C09107=1059.255,344.994,392.279,173.812,36.431,156.854
C09108=1059.262,345.241,392.243,173.816,36.436,156.855
C09109=1059.268,345.487,392.207,173.819,36.441,156.856
C09110=1059.276,345.733,392.171,173.824,36.446,156.857
C09111=1059.282,345.979,392.135,173.828,36.451,156.859
C09112=1059.289,346.224,392.098,173.832,36.455,156.860
C09113=1059.296,346.470,392.063,173.836,36.460,156.861
C09114=1059.302,346.716,392.026,173.841,36.466,156.862
C09115=1059.308,346.961,391.990,173.844,36.471,156.863
C09116=1059.315,347.208,391.954,173.848,36.476,156.864
C09117=1059.323,347.455,391.918,173.853,36.480,156.865
C09118=1059.329,347.702,391.882,173.856,36.485,156.866
C09119=1059.336,347.950,391.845,173.861,36.490,156.868
C09120=1059.343,348.196,391.809,173.865,36.495,156.869
C09121=1059.350,348.444,391.772,173.869,36.500,156.870
C09122=1059.356,348.690,391.735,173.873,36.506,156.871
C09123=1059.363,348.938,391.698,173.878,36.511,156.872
C09124=1059.371,349.185,391.662,173.881,36.516,156.873
C09125=1059.377,349.433,391.626,173.886,36.521,156.875
C09126=1059.384,349.680,391.589,173.890,36.526,156.876
C09127=1059.391,349.928,391.552,173.895,36.531,156.877
C09128=1059.398,350.174,391.517,173.898,36.536,156.878
C09129=1059.405,350.421,391.479,173.903,36.541,156.879
C09130=1059.411,350.668,391.443,173.907,36.547,156.881
C09131=1059.418,350.916,391.406,173.911,36.552,156.882
C09132=1059.425,351.163,391.370,173.916,36.557,156.883
C09133=1059.433,351.410,391.332,173.920,36.562,156.884
C09134=1059.439,351.657,391.296,173.925,36.567,156.885
C09135=1059.446,351.905,391.259,173.928,36.572,156.886
C09136=1059.453,352.151,391.222,173.933,36.578,156.888
C09137=1059.459,352.399,391.185,173.937,36.583,156.889
C09138=1059.466,352.647,391.148,173.941,36.588,156.890
C09139=1059.473,352.893,391.111,173.945,36.593,156.891
C09140=1059.480,353.141,391.074,173.950,36.598,156.893
C09141=1059.487,353.387,391.037,173.955,36.603,156.894
C09142=1059.494,353.635,391.000,173.959,36.609,156.895
C09143=1059.500,353.882,390.963,173.963,36.614,156.896
C09144=1059.507,354.129,390.926,173.967,36.619,156.897
C09145=1059.514,354.377,390.889,173.972,36.625,156.899
C09146=1059.521,354.623,390.852,173.976,36.630,156.900
C09147=1059.528,354.871,390.815,173.980,36.635,156.901
C09148=1059.535,355.118,390.777,173.985,36.640,156.902
C09149=1059.542,355.364,390.740,173.989,36.646,156.904
C09150=1059.549,355.612,390.703,173.994,36.651,156.905
C09151=1059.556,355.859,390.666,173.998,36.656,156.906
C09152=1059.563,356.106,390.629,174.002,36.662,156.907
C09153=1059.570,356.353,390.592,174.007,36.667,156.909
C09154=1059.577,356.601,390.554,174.012,36.672,156.910
C09155=1059.584,356.848,390.517,174.015,36.678,156.911
C09156=1059.591,357.094,390.480,174.020,36.683,156.912
C09157=1059.598,357.342,390.443,174.025,36.688,156.914
C09158=1059.605,357.589,390.405,174.029,36.694,156.915
C09159=1059.612,357.836,390.368,174.033,36.699,156.916
C09160=1059.619,358.083,390.330,174.038,36.705,156.917
C09161=1059.626,358.330,390.293,174.042,36.710,156.919
C09162=1059.633,358.577,390.256,174.047,36.715,156.920
C09163=1059.640,358.824,390.217,174.052,36.721,156.921
C09164=1059.647,359.071,390.180,174.056,36.726,156.923
C09165=1059.654,359.320,390.142,174.060,36.732,156.924
C09166=1059.661,359.569,390.104,174.065,36.737,156.925
C09167=1059.667,359.818,390.067,174.070,36.743,156.927
C09168=1059.675,360.067,390.028,174.074,36.749,156.928
C09169=1059.682,360.313,389.991,174.079,36.754,156.929
C09170=1059.689,360.560,389.953,174.083,36.760,156.930
C09171=1059.696,360.807,389.916,174.087,36.765,156.932
C09172=1059.703,361.055,389.877,174.092,36.770,156.933
C09173=1059.710,361.302,389.840,174.097,36.776,156.934
C09174=1059.717,361.549,389.802,174.102,36.781,156.936
C09175=1059.725,361.796,389.764,174.106,36.787,156.937
C09176=1059.731,362.043,389.726,174.110,36.793,156.938
C09177=1059.739,362.290,389.689,174.115,36.799,156.940
C09178=1059.746,362.536,389.651,174.120,36.804,156.941
C09179=1059.752,362.783,389.613,174.124,36.810,156.942
C09180=1059.759,363.031,389.575,174.129,36.815,156.944
C09181=1059.767,363.277,389.537,174.134,36.821,156.945
C09182=1059.773,363.525,389.499,174.139,36.826,156.946
C09183=1059.781,363.772,389.461,174.143,36.832,156.948
C09184=1059.788,364.018,389.423,174.147,36.838,156.949
C09185=1059.795,364.266,389.385,174.152,36.844,156.950
C09186=1059.802,364.512,389.346,174.157,36.849,156.952
C09187=1059.809,364.760,389.308,174.162,36.855,156.953
C09188=1059.815,365.006,389.270,174.166,36.861,156.954
C09189=1059.823,365.253,389.231,174.171,36.866,156.956
C09190=1059.830,365.500,389.193,174.176,36.873,156.957
C09191=1059.837,365.747,389.155,174.180,36.878,156.959
C09192=1059.844,365.994,389.116,174.185,36.884,156.960
C09193=1059.851,366.241,389.079,174.190,36.890,156.961
C09194=1059.858,366.488,389.040,174.194,36.896,156.963
C09195=1059.866,366.734,389.001,174.199,36.901,156.964
C09196=1059.873,366.982,388.963,174.204,36.907,156.966
C09197=1059.879,367.229,388.924,174.209,36.913,156.967
C09198=1059.887,367.476,388.886,174.214,36.919,156.968
C09199=1059.894,367.722,388.847,174.219,36.925,156.970
C09200=1059.901,367.969,388.809,174.223,36.931,156.971
C09201=1059.908,368.216,388.770,174.228,36.937,156.973
C09202=1059.915,368.463,388.732,174.232,36.942,156.974
C09203=1059.922,368.710,388.694,174.237,36.948,156.975
C09204=1059.930,368.957,388.654,174.242,36.954,156.977
C09205=1059.936,369.204,388.616,174.247,36.960,156.978
C09206=1059.944,369.451,388.577,174.252,36.966,156.980
C09207=1059.951,369.697,388.539,174.257,36.972,156.981
C09208=1059.958,369.944,388.500,174.262,36.978,156.983
C09209=1059.966,370.192,388.461,174.267,36.984,156.984
C09210=1059.973,370.438,388.422,174.271,36.990,156.985
C09211=1059.980,370.684,388.383,174.276,36.996,156.987
C09212=1059.987,370.931,388.344,174.281,37.002,156.988
C09213=1059.995,371.179,388.305,174.286,37.008,156.990
C09214=1060.002,371.425,388.267,174.291,37.014,156.991
C09215=1060.009,371.672,388.228,174.296,37.020,156.993
C09216=1060.016,371.919,388.189,174.301,37.026,156.994
C09217=1060.024,372.165,388.150,174.306,37.032,156.996
C09218=1060.031,372.412,388.111,174.311,37.038,156.997
C09219=1060.039,372.660,388.072,174.316,37.044,156.999
C09220=1060.046,372.906,388.032,174.321,37.050,157.000
C09221=1060.053,373.173,387.990,174.326,37.057,157.002
C09222=1060.060,373.440,387.948,174.332,37.064,157.003
C09223=1060.069,373.707,387.906,174.337,37.071,157.005
C09224=1060.077,373.974,387.863,174.342,37.077,157.007
C09225=1060.084,374.221,387.824,174.347,37.083,157.008
C09226=1060.091,374.468,387.785,174.352,37.090,157.010
C09227=1060.098,374.714,387.745,174.357,37.096,157.011
C09228=1060.106,374.962,387.706,174.362,37.102,157.013
C09229=1060.113,375.208,387.666,174.367,37.109,157.014
C09230=1060.120,375.454,387.627,174.372,37.115,157.016
C09231=1060.127,375.702,387.588,174.377,37.121,157.017
C09232=1060.134,375.948,387.548,174.382,37.127,157.019
C09233=1060.142,376.195,387.509,174.388,37.134,157.020
C09234=1060.149,376.442,387.469,174.394,37.140,157.022
C09235=1060.157,376.689,387.429,174.399,37.146,157.023
C09236=1060.164,376.935,387.390,174.404,37.152,157.025
C09237=1060.171,377.182,387.351,174.409,37.159,157.027
C09238=1060.178,377.429,387.311,174.414,37.166,157.028
C09239=1060.186,377.675,387.271,174.419,37.172,157.030
C09240=1060.193,377.922,387.232,174.424,37.178,157.031
C09241=1060.201,378.169,387.192,174.429,37.185,157.033
C09242=1060.208,378.415,387.152,174.434,37.191,157.034
C09243=1060.216,378.662,387.112,174.439,37.197,157.036
C09244=1060.223,378.908,387.073,174.444,37.204,157.038
C09245=1060.231,379.155,387.033,174.451,37.211,157.039
C09246=1060.238,379.402,386.993,174.456,37.217,157.041
C09247=1060.245,379.648,386.953,174.461,37.223,157.042
C09248=1060.253,379.895,386.913,174.466,37.230,157.044
C09249=1060.261,380.142,386.873,174.471,37.236,157.045
C09250=1060.267,380.388,386.833,174.476,37.243,157.047
C09251=1060.275,380.635,386.793,174.482,37.249,157.049
C09252=1060.283,380.882,386.753,174.487,37.256,157.050
C09253=1060.290,381.128,386.714,174.492,37.262,157.052
C09254=1060.297,381.375,386.673,174.498,37.270,157.054
C09255=1060.304,381.621,386.633,174.503,37.276,157.055
C09256=1060.312,381.868,386.593,174.508,37.283,157.057
C09257=1060.319,382.114,386.552,174.514,37.289,157.059
C09258=1060.326,382.361,386.512,174.519,37.296,157.060
C09259=1060.334,382.608,386.472,174.524,37.303,157.062
C09260=1060.341,382.854,386.431,174.530,37.309,157.064
C09261=1060.349,383.101,386.391,174.535,37.316,157.065
C09262=1060.356,383.347,386.351,174.541,37.323,157.067
C09263=1060.363,383.594,386.311,174.546,37.330,157.069
C09264=1060.371,383.840,386.270,174.551,37.337,157.070
C09265=1060.378,384.087,386.229,174.557,37.344,157.072
C09266=1060.386,384.333,386.189,174.562,37.350,157.074
C09267=1060.394,384.580,386.149,174.568,37.357,157.075
C09268=1060.401,384.826,386.108,174.573,37.364,157.077
C09269=1060.409,385.073,386.067,174.578,37.371,157.079
C09270=1060.417,385.320,386.027,174.585,37.378,157.081
C09271=1060.424,385.566,385.986,174.590,37.384,157.082
C09272=1060.431,385.812,385.946,174.595,37.391,157.084
C09273=1060.438,386.059,385.905,174.600,37.398,157.086
C09274=1060.446,386.305,385.865,174.607,37.405,157.087
C09275=1060.454,386.552,385.824,174.612,37.412,157.089
C09276=1060.462,386.798,385.783,174.617,37.419,157.091
C09277=1060.471,387.097,385.733,174.625,37.428,157.093
C09278=1060.481,387.395,385.684,174.631,37.436,157.095
C09279=1060.490,387.693,385.635,174.638,37.445,157.097
C09280=1060.499,387.992,385.585,174.644,37.453,157.099
C09281=1060.507,388.238,385.545,174.650,37.460,157.101
C09282=1060.514,388.484,385.503,174.656,37.467,157.103
C09283=1060.522,388.731,385.463,174.661,37.474,157.105
C09284=1060.529,388.977,385.421,174.667,37.481,157.107
C09285=1060.537,389.224,385.381,174.673,37.488,157.108
C09286=1060.545,389.470,385.340,174.679,37.495,157.110
C09287=1060.553,389.716,385.299,174.684,37.502,157.112
C09288=1060.560,389.962,385.257,174.691,37.509,157.114
C09289=1060.568,390.209,385.216,174.696,37.517,157.116
C09290=1060.576,390.455,385.175,174.701,37.524,157.117
C09291=1060.583,390.702,385.134,174.708,37.531,157.119
C09292=1060.592,390.948,385.092,174.713,37.539,157.121
C09293=1060.599,391.195,385.051,174.719,37.546,157.123
C09294=1060.606,391.441,385.010,174.725,37.553,157.125
C09295=1060.615,391.687,384.968,174.731,37.560,157.126
C09296=1060.622,391.934,384.927,174.737,37.568,157.128
C09297=1060.630,392.180,384.885,174.742,37.575,157.130
C09298=1060.637,392.426,384.844,174.748,37.582,157.132
C09299=1060.646,392.673,384.802,174.754,37.590,157.134
C09300=1060.653,392.919,384.761,174.760,37.597,157.136
C09301=1060.661,393.165,384.719,174.765,37.604,157.138
C09302=1060.668,393.412,384.678,174.772,37.612,157.140
C09303=1060.676,393.658,384.636,174.777,37.620,157.141
C09304=1060.684,393.904,384.594,174.784,37.627,157.143
C09305=1060.692,394.150,384.552,174.790,37.635,157.145
C09306=1060.699,394.397,384.511,174.796,37.642,157.147
C09307=1060.707,394.643,384.469,174.802,37.650,157.149
C09308=1060.715,394.889,384.427,174.807,37.657,157.151
C09309=1060.723,395.135,384.385,174.814,37.665,157.153
C09310=1060.730,395.382,384.344,174.819,37.672,157.155
C09311=1060.738,395.629,384.301,174.826,37.680,157.157
C09312=1060.746,395.875,384.259,174.831,37.688,157.159
C09313=1060.753,396.121,384.217,174.838,37.695,157.161
C09314=1060.762,396.367,384.175,174.844,37.703,157.163
C09315=1060.769,396.613,384.133,174.850,37.711,157.165
C09316=1060.777,396.860,384.091,174.856,37.718,157.167
C09317=1060.786,397.106,384.050,174.862,37.726,157.169
C09318=1060.794,397.352,384.007,174.868,37.734,157.171
C09319=1060.801,397.598,383.965,174.875,37.741,157.173
C09320=1060.809,397.845,383.922,174.880,37.749,157.175
C09321=1060.817,398.091,383.880,174.887,37.758,157.177
C09322=1060.825,398.337,383.837,174.892,37.765,157.179
C09323=1060.833,398.583,383.795,174.899,37.773,157.181
C09324=1060.841,398.830,383.753,174.906,37.781,157.183
C09325=1060.849,399.075,383.710,174.911,37.789,157.185
C09326=1060.857,399.322,383.668,174.918,37.797,157.187
C09327=1060.864,399.568,383.626,174.924,37.805,157.189
C09328=1060.872,399.814,383.583,174.931,37.813,157.191
C09329=1060.880,400.060,383.541,174.937,37.821,157.193
C09330=1060.888,400.306,383.498,174.943,37.829,157.195
C09331=1060.897,400.553,383.455,174.950,37.837,157.197
C09332=1060.905,400.798,383.413,174.955,37.845,157.199
C09333=1060.915,401.114,383.358,174.963,37.855,157.202
C09334=1060.925,401.430,383.304,174.973,37.865,157.205
C09335=1060.935,401.745,383.248,174.981,37.876,157.207
C09336=1060.946,402.060,383.194,174.989,37.886,157.210
C09337=1060.953,402.307,383.151,174.995,37.894,157.212
C09338=1060.962,402.553,383.108,175.001,37.902,157.214
C09339=1060.970,402.798,383.065,175.008,37.911,157.216
C09340=1060.977,403.045,383.022,175.014,37.919,157.219
C09341=1060.986,403.291,382.979,175.021,37.927,157.221
C09342=1060.994,403.537,382.936,175.028,37.935,157.223
C09343=1061.002,403.784,382.892,175.034,37.944,157.225
C09344=1061.010,404.029,382.850,175.040,37.952,157.227
C09345=1061.018,404.275,382.806,175.047,37.960,157.229
C09346=1061.026,404.521,382.763,175.054,37.969,157.232
C09347=1061.035,404.767,382.720,175.061,37.977,157.234
C09348=1061.042,405.014,382.676,175.067,37.986,157.236
C09349=1061.051,405.260,382.633,175.074,37.994,157.238
C09350=1061.059,405.506,382.590,175.080,38.002,157.240
C09351=1061.067,405.752,382.547,175.086,38.011,157.243
C09352=1061.075,405.999,382.503,175.093,38.020,157.245
C09353=1061.083,406.244,382.459,175.100,38.028,157.247
C09354=1061.092,406.490,382.416,175.107,38.037,157.249
C09355=1061.099,406.737,382.372,175.114,38.045,157.252
C09356=1061.107,406.982,382.328,175.121,38.054,157.254
C09357=1061.116,407.229,382.285,175.127,38.063,157.256
C09358=1061.124,407.475,382.241,175.134,38.071,157.259
C09359=1061.132,407.720,382.197,175.141,38.080,157.261
C09360=1061.140,407.967,382.154,175.148,38.089,157.263
C09361=1061.148,408.212,382.109,175.155,38.097,157.265
C09362=1061.157,408.458,382.066,175.162,38.106,157.268
C09363=1061.165,408.704,382.022,175.169,38.115,157.270
C09364=1061.173,408.951,381.978,175.175,38.123,157.272
C09365=1061.181,409.196,381.935,175.182,38.132,157.275
C09366=1061.190,409.442,381.890,175.189,38.141,157.277
C09367=1061.198,409.689,381.846,175.196,38.150,157.280
C09368=1061.206,409.935,381.802,175.203,38.159,157.282
C09369=1061.215,410.180,381.758,175.210,38.168,157.284
C09370=1061.223,410.426,381.714,175.217,38.177,157.287
C09371=1061.231,410.672,381.670,175.225,38.186,157.289
C09372=1061.240,410.918,381.626,175.232,38.195,157.291
C09373=1061.248,411.164,381.582,175.239,38.204,157.294
C09374=1061.256,411.410,381.538,175.246,38.213,157.296
C09375=1061.265,411.656,381.493,175.253,38.222,157.299
C09376=1061.274,411.902,381.449,175.260,38.231,157.301
C09377=1061.282,412.147,381.405,175.268,38.240,157.303
C09378=1061.290,412.394,381.360,175.275,38.249,157.306
C09379=1061.298,412.640,381.316,175.282,38.258,157.308
C09380=1061.308,412.886,381.272,175.289,38.267,157.311
C09381=1061.316,413.131,381.227,175.296,38.277,157.313
C09382=1061.324,413.377,381.182,175.304,38.286,157.316
C09383=1061.333,413.623,381.138,175.311,38.295,157.318
C09384=1061.342,413.868,381.094,175.318,38.304,157.321
C09385=1061.350,414.115,381.049,175.326,38.314,157.323
C09386=1061.359,414.360,381.004,175.333,38.323,157.326
C09387=1061.368,414.606,380.959,175.341,38.332,157.328
C09388=1061.376,414.852,380.914,175.348,38.342,157.331
C09389=1061.389,415.252,380.841,175.360,38.357,157.335
C09390=1061.404,415.652,380.768,175.373,38.373,157.339
C09391=1061.417,416.053,380.695,175.385,38.388,157.343
C09392=1061.431,416.453,380.621,175.397,38.404,157.348
C09393=1061.439,416.698,380.576,175.405,38.413,157.350
C09394=1061.448,416.943,380.531,175.412,38.423,157.353
C09395=1061.457,417.189,380.486,175.420,38.432,157.355
C09396=1061.465,417.435,380.441,175.428,38.442,157.358
C09397=1061.474,417.681,380.396,175.435,38.452,157.361
C09398=1061.483,417.927,380.350,175.443,38.462,157.363
C09399=1061.492,418.172,380.305,175.450,38.472,157.366
C09400=1061.501,418.418,380.260,175.459,38.481,157.369
C09401=1061.509,418.664,380.214,175.466,38.491,157.371
C09402=1061.518,418.910,380.168,175.474,38.501,157.374
C09403=1061.526,419.155,380.123,175.482,38.511,157.377
C09404=1061.535,419.401,380.078,175.490,38.520,157.379
C09405=1061.544,419.646,380.032,175.498,38.530,157.382
C09406=1061.554,419.892,379.986,175.506,38.540,157.385
C09407=1061.562,420.138,379.940,175.514,38.551,157.388
C09408=1061.571,420.384,379.895,175.521,38.561,157.390
C09409=1061.585,420.795,379.818,175.535,38.577,157.395
C09410=1061.600,421.207,379.741,175.548,38.594,157.400
C09411=1061.615,421.618,379.664,175.563,38.611,157.404
C09412=1061.629,422.030,379.587,175.576,38.629,157.409
C09413=1061.639,422.275,379.541,175.584,38.639,157.412
C09414=1061.647,422.521,379.495,175.593,38.649,157.415
C09415=1061.656,422.767,379.449,175.600,38.660,157.418
C09416=1061.665,423.012,379.402,175.609,38.670,157.421
C09417=1061.674,423.258,379.356,175.617,38.680,157.424
C09418=1061.683,423.504,379.310,175.626,38.691,157.426
C09419=1061.692,423.750,379.263,175.633,38.701,157.429
C09420=1061.701,423.995,379.217,175.642,38.711,157.432
C09421=1061.710,424.240,379.170,175.651,38.722,157.435
C09422=1061.719,424.486,379.124,175.659,38.733,157.438
C09423=1061.728,424.731,379.077,175.668,38.743,157.441
C09424=1061.737,424.976,379.031,175.675,38.754,157.444
C09425=1061.747,425.222,378.985,175.684,38.765,157.447
C09426=1061.755,425.468,378.938,175.693,38.775,157.450
C09427=1061.765,425.713,378.892,175.701,38.786,157.453
C09428=1061.773,425.958,378.845,175.710,38.797,157.456
C09429=1061.783,426.204,378.798,175.719,38.807,157.459
C09430=1061.792,426.449,378.751,175.727,38.818,157.462
C09431=1061.801,426.695,378.704,175.736,38.828,157.465
C09432=1061.811,426.940,378.657,175.745,38.839,157.468
C09433=1061.819,427.185,378.611,175.754,38.851,157.471
C09434=1061.828,427.432,378.563,175.762,38.861,157.474
C09435=1061.838,427.676,378.517,175.771,38.872,157.477
C09436=1061.847,427.921,378.469,175.780,38.884,157.480
C09437=1061.856,428.167,378.422,175.789,38.894,157.483
C09438=1061.865,428.412,378.375,175.798,38.906,157.487
C09439=1061.875,428.658,378.327,175.806,38.916,157.490
C09440=1061.884,428.903,378.281,175.815,38.928,157.493
C09441=1061.897,429.244,378.215,175.828,38.943,157.497
C09442=1061.909,429.585,378.149,175.840,38.959,157.502
C09443=1061.923,429.926,378.083,175.853,38.974,157.506
C09444=1061.935,430.266,378.017,175.865,38.990,157.511
C09445=1061.945,430.512,377.969,175.875,39.001,157.514
C09446=1061.954,430.758,377.922,175.884,39.013,157.517
C09447=1061.963,431.002,377.874,175.893,39.024,157.520
C09448=1061.972,431.248,377.826,175.902,39.036,157.524
C09449=1061.982,431.494,377.778,175.911,39.047,157.527
C09450=1061.991,431.738,377.730,175.921,39.059,157.530
C09451=1062.001,431.984,377.682,175.931,39.070,157.534
C09452=1062.010,432.229,377.635,175.940,39.082,157.537
C09453=1062.019,432.473,377.587,175.950,39.093,157.540
C09454=1062.029,432.719,377.539,175.959,39.105,157.543
C09455=1062.038,432.964,377.490,175.968,39.117,157.547
C09456=1062.048,433.210,377.442,175.978,39.128,157.550
C09457=1062.058,433.455,377.394,175.987,39.141,157.554
C09458=1062.067,433.699,377.346,175.996,39.152,157.557
C09459=1062.076,433.944,377.298,176.007,39.164,157.560
C09460=1062.086,434.189,377.249,176.016,39.176,157.564
C09461=1062.096,434.434,377.201,176.026,39.188,157.567
C09462=1062.105,434.679,377.152,176.035,39.200,157.571
C09463=1062.115,434.925,377.104,176.046,39.212,157.574
C09464=1062.125,435.170,377.056,176.055,39.224,157.578
C09465=1062.134,435.415,377.007,176.065,39.236,157.581
C09466=1062.143,435.660,376.958,176.074,39.248,157.585
C09467=1062.153,435.905,376.910,176.085,39.260,157.588
C09468=1062.163,436.150,376.861,176.095,39.272,157.592
C09469=1062.173,436.395,376.813,176.105,39.285,157.595
C09470=1062.183,436.639,376.763,176.115,39.297,157.599
C09471=1062.193,436.884,376.715,176.125,39.309,157.603
C09472=1062.202,437.129,376.666,176.135,39.321,157.606
C09473=1062.213,437.375,376.618,176.145,39.334,157.610
C09474=1062.223,437.619,376.568,176.156,39.346,157.613
C09475=1062.232,437.865,376.519,176.165,39.359,157.617
C09476=1062.242,438.109,376.470,176.176,39.371,157.621
C09477=1062.252,438.355,376.421,176.186,39.384,157.624
C09478=1062.262,438.599,376.371,176.197,39.396,157.628
C09479=1062.271,438.844,376.323,176.206,39.409,157.632
C09480=1062.281,439.089,376.273,176.217,39.422,157.636
C09481=1062.291,439.334,376.223,176.227,39.434,157.639
C09482=1062.301,439.578,376.174,176.238,39.447,157.643
C09483=1062.311,439.823,376.125,176.249,39.460,157.647
C09484=1062.321,440.069,376.075,176.259,39.472,157.651
C09485=1062.331,440.313,376.026,176.270,39.485,157.654
C09486=1062.341,440.558,375.976,176.281,39.498,157.658
C09487=1062.351,440.803,375.927,176.291,39.511,157.662
C09488=1062.361,441.047,375.877,176.301,39.524,157.666
C09489=1062.371,441.292,375.826,176.312,39.537,157.670
C09490=1062.381,441.536,375.777,176.323,39.550,157.674
C09491=1062.391,441.782,375.727,176.335,39.564,157.678
C09492=1062.401,442.026,375.678,176.346,39.577,157.682
C09493=1062.412,442.271,375.627,176.356,39.590,157.686
C09494=1062.422,442.516,375.577,176.367,39.603,157.690
C09495=1062.432,442.760,375.527,176.378,39.616,157.693
C09496=1062.443,443.005,375.477,176.389,39.630,157.698
C09497=1062.453,443.260,375.424,176.400,39.644,157.702
C09498=1062.464,443.514,375.372,176.413,39.658,157.706
C09499=1062.474,443.769,375.319,176.424,39.672,157.710
C09500=1062.486,444.024,375.267,176.436,39.685,157.714
C09501=1062.495,444.268,375.217,176.447,39.699,157.718
C09502=1062.505,444.513,375.166,176.459,39.713,157.723
C09503=1062.516,444.758,375.116,176.470,39.726,157.727
C09504=1062.526,445.002,375.065,176.481,39.740,157.731
C09505=1062.537,445.247,375.014,176.493,39.754,157.735
C09506=1062.548,445.492,374.964,176.505,39.767,157.739
C09507=1062.557,445.736,374.913,176.516,39.781,157.743
C09508=1062.567,445.980,374.862,176.528,39.795,157.748
C09509=1062.579,446.224,374.811,176.539,39.809,157.752
C09510=1062.589,446.469,374.760,176.552,39.823,157.756
C09511=1062.599,446.714,374.709,176.563,39.837,157.760
C09512=1062.610,446.957,374.658,176.575,39.851,157.765
C09513=1062.621,447.202,374.607,176.587,39.865,157.769
C09514=1062.632,447.445,374.556,176.599,39.879,157.773
C09515=1062.643,447.689,374.506,176.610,39.893,157.777
C09516=1062.655,447.933,374.457,176.622,39.907,157.782
C09517=1062.668,448.177,374.406,176.635,39.920,157.786
C09518=1062.683,448.421,374.358,176.647,39.933,157.790
C09519=1062.697,448.665,374.311,176.659,39.946,157.794
C09520=1062.714,448.910,374.263,176.672,39.958,157.798
C09521=1062.730,449.155,374.217,176.684,39.971,157.802
C09522=1062.749,449.400,374.170,176.697,39.983,157.806
C09523=1062.767,449.646,374.125,176.710,39.994,157.809
C09524=1062.788,449.891,374.081,176.722,40.006,157.813
C09525=1062.452,449.899,373.808,176.715,40.125,157.846
C09526=1062.433,449.654,373.853,176.702,40.114,157.842
C09527=1062.414,449.409,373.898,176.689,40.102,157.838
C09528=1062.395,449.163,373.944,176.677,40.090,157.834
C09529=1062.379,448.919,373.990,176.664,40.078,157.830
C09530=1062.362,448.673,374.037,176.652,40.065,157.826
C09531=1062.347,448.429,374.086,176.639,40.052,157.822
C09532=1062.332,448.185,374.134,176.627,40.039,157.818
C09533=1062.319,447.941,374.183,176.615,40.026,157.814
C09534=1062.307,447.697,374.233,176.602,40.013,157.810
C09535=1062.295,447.453,374.283,176.591,39.999,157.806
C09536=1062.284,447.210,374.334,176.578,39.985,157.801
C09537=1062.274,446.967,374.385,176.567,39.971,157.797
C09538=1062.263,446.723,374.436,176.555,39.957,157.793
C09539=1062.252,446.478,374.487,176.542,39.943,157.789
C09540=1062.242,446.233,374.538,176.531,39.929,157.784
C09541=1062.231,445.989,374.589,176.519,39.916,157.780
C09542=1062.221,445.745,374.640,176.507,39.902,157.776
C09543=1062.210,445.500,374.691,176.496,39.888,157.772
C09544=1062.199,445.256,374.742,176.484,39.874,157.767
C09545=1062.189,445.011,374.792,176.473,39.860,157.763
C09546=1062.179,444.771,374.842,176.462,39.847,157.759
C09547=1062.169,444.530,374.892,176.449,39.834,157.755
C09548=1062.158,444.290,374.941,176.438,39.820,157.751
C09549=1062.148,444.050,374.991,176.427,39.807,157.747
C09550=1062.138,443.810,375.041,176.416,39.794,157.743
C09551=1062.128,443.570,375.090,176.405,39.780,157.739
C09552=1062.118,443.331,375.139,176.394,39.767,157.735
C09553=1062.108,443.091,375.189,176.383,39.754,157.731
C09554=1062.097,442.846,375.240,176.371,39.741,157.727
C09555=1062.087,442.602,375.289,176.360,39.728,157.723
C09556=1062.077,442.357,375.340,176.349,39.715,157.719
C09557=1062.067,442.112,375.389,176.339,39.702,157.715
C09558=1062.057,441.867,375.440,176.328,39.688,157.711
C09559=1062.046,441.623,375.490,176.317,39.675,157.707
C09560=1062.037,441.378,375.540,176.306,39.662,157.703
C09561=1062.026,441.133,375.589,176.295,39.649,157.699
C09562=1062.017,440.888,375.639,176.284,39.636,157.695
C09563=1062.006,440.643,375.689,176.273,39.624,157.692
C09564=1061.996,440.400,375.739,176.263,39.610,157.688
C09565=1061.986,440.154,375.789,176.252,39.597,157.684
C09566=1061.976,439.910,375.838,176.241,39.585,157.680
C09567=1061.966,439.664,375.888,176.230,39.572,157.676
C09568=1061.956,439.419,375.937,176.220,39.559,157.673
C09569=1061.946,439.175,375.986,176.209,39.547,157.669
C09570=1061.936,438.930,376.036,176.199,39.534,157.665
C09571=1061.926,438.685,376.086,176.189,39.522,157.661
C09572=1061.916,438.440,376.134,176.178,39.509,157.658
C09573=1061.906,438.195,376.184,176.167,39.496,157.654
C09574=1061.897,437.950,376.233,176.157,39.484,157.650
C09575=1061.887,437.706,376.282,176.147,39.471,157.646
C09576=1061.877,437.461,376.331,176.137,39.459,157.643
C09577=1061.867,437.215,376.381,176.126,39.447,157.639
C09578=1061.857,436.970,376.429,176.116,39.434,157.636
C09579=1061.847,436.725,376.478,176.106,39.422,157.632
C09580=1061.837,436.481,376.527,176.096,39.410,157.629
C09581=1061.828,436.236,376.576,176.085,39.398,157.625
C09582=1061.818,435.991,376.624,176.076,39.386,157.621
C09583=1061.808,435.746,376.673,176.066,39.374,157.618
C09584=1061.798,435.501,376.722,176.056,39.362,157.614
C09585=1061.788,435.256,376.770,176.046,39.350,157.611
C09586=1061.778,435.011,376.819,176.035,39.337,157.607
C09587=1061.768,434.766,376.867,176.026,39.326,157.604
C09588=1061.759,434.521,376.916,176.016,39.314,157.600
C09589=1061.749,434.276,376.964,176.007,39.302,157.597
C09590=1061.741,434.030,377.012,175.996,39.290,157.593
C09591=1061.731,433.786,377.061,175.987,39.278,157.590
C09592=1061.721,433.541,377.109,175.978,39.266,157.587
C09593=1061.711,433.296,377.158,175.968,39.255,157.583
C09594=1061.702,433.050,377.206,175.958,39.243,157.580
C09595=1061.692,432.805,377.254,175.948,39.231,157.576
C09596=1061.683,432.560,377.302,175.939,39.220,157.573
C09597=1061.674,432.315,377.350,175.930,39.208,157.570
C09598=1061.664,432.070,377.398,175.920,39.196,157.566
C09599=1061.654,431.825,377.447,175.911,39.185,157.563
C09600=1061.646,431.580,377.494,175.901,39.173,157.560
C09601=1061.636,431.334,377.542,175.892,39.161,157.556
C09602=1061.627,431.088,377.590,175.882,39.150,157.553
C09603=1061.618,430.844,377.638,175.873,39.139,157.550
C09604=1061.608,430.599,377.686,175.864,39.127,157.546
C09605=1061.598,430.353,377.733,175.855,39.116,157.543
C09606=1061.586,430.010,377.799,175.842,39.100,157.539
C09607=1061.573,429.668,377.866,175.829,39.085,157.534
C09608=1061.560,429.325,377.932,175.817,39.069,157.530
C09609=1061.547,428.982,377.998,175.804,39.054,157.525
C09610=1061.537,428.737,378.045,175.795,39.042,157.522
C09611=1061.528,428.492,378.093,175.786,39.031,157.519
C09612=1061.518,428.246,378.141,175.777,39.020,157.516
C09613=1061.510,428.001,378.187,175.768,39.010,157.513
C09614=1061.499,427.755,378.235,175.759,38.998,157.510
C09615=1061.491,427.510,378.281,175.750,38.987,157.507
C09616=1061.481,427.264,378.329,175.742,38.977,157.504
C09617=1061.472,427.020,378.376,175.733,38.965,157.500
C09618=1061.463,426.774,378.423,175.724,38.955,157.497
C09619=1061.454,426.528,378.470,175.715,38.944,157.494
C09620=1061.445,426.283,378.517,175.706,38.933,157.491
C09621=1061.436,426.038,378.563,175.698,38.923,157.488
C09622=1061.426,425.792,378.610,175.689,38.912,157.485
C09623=1061.418,425.546,378.657,175.680,38.901,157.482
C09624=1061.408,425.302,378.703,175.672,38.891,157.479
C09625=1061.399,425.056,378.751,175.663,38.880,157.476
C09626=1061.390,424.810,378.797,175.654,38.870,157.473
C09627=1061.381,424.565,378.843,175.645,38.859,157.470
C09628=1061.372,424.320,378.890,175.637,38.849,157.467
C09629=1061.363,424.074,378.936,175.629,38.838,157.464
C09630=1061.353,423.828,378.983,175.621,38.827,157.462
C09631=1061.345,423.583,379.029,175.612,38.817,157.459
C09632=1061.336,423.338,379.076,175.603,38.807,157.456
C09633=1061.327,423.092,379.121,175.595,38.796,157.453
C09634=1061.318,422.846,379.168,175.587,38.786,157.450
C09635=1061.309,422.601,379.214,175.579,38.776,157.447
C09636=1061.300,422.356,379.261,175.570,38.765,157.444
C09637=1061.291,422.110,379.306,175.562,38.755,157.441
C09638=1061.283,421.864,379.353,175.554,38.745,157.439
C09639=1061.273,421.619,379.399,175.546,38.735,157.436
C09640=1061.264,421.373,379.444,175.537,38.724,157.433
C09641=1061.256,421.128,379.491,175.530,38.714,157.430
C09642=1061.247,420.882,379.536,175.521,38.704,157.427
C09643=1061.238,420.636,379.583,175.514,38.694,157.424
C09644=1061.229,420.391,379.629,175.505,38.684,157.422
C09645=1061.220,420.145,379.674,175.497,38.674,157.419
C09646=1061.211,419.899,379.720,175.489,38.664,157.416
C09647=1061.203,419.653,379.766,175.481,38.654,157.413
C09648=1061.194,419.408,379.811,175.474,38.644,157.411
C09649=1061.185,419.162,379.857,175.465,38.634,157.408
C09650=1061.177,418.917,379.902,175.457,38.625,157.405
C09651=1061.168,418.671,379.947,175.449,38.615,157.403
C09652=1061.159,418.425,379.993,175.441,38.605,157.400
C09653=1061.150,418.179,380.038,175.434,38.595,157.397
C09654=1061.141,417.934,380.083,175.425,38.586,157.395
C09655=1061.133,417.688,380.129,175.418,38.576,157.392
C09656=1061.124,417.442,380.175,175.410,38.566,157.389
C09657=1061.116,417.197,380.220,175.403,38.556,157.387
C09658=1061.107,416.951,380.265,175.395,38.547,157.384
C09659=1061.098,416.705,380.311,175.387,38.538,157.381
C09660=1061.090,416.460,380.355,175.380,38.528,157.379
C09661=1061.081,416.214,380.400,175.372,38.518,157.376
C09662=1061.069,415.891,380.460,175.362,38.506,157.373
C09663=1061.058,415.569,380.519,175.352,38.493,157.369
C09664=1061.047,415.247,380.578,175.342,38.481,157.366
C09665=1061.036,414.924,380.637,175.332,38.469,157.363
C09666=1061.028,414.678,380.682,175.325,38.459,157.360
C09667=1061.019,414.433,380.727,175.318,38.450,157.358
C09668=1061.010,414.186,380.772,175.309,38.440,157.355
C09669=1061.002,413.941,380.817,175.302,38.431,157.352
C09670=1060.993,413.695,380.861,175.295,38.422,157.350
C09671=1060.985,413.449,380.905,175.287,38.413,157.347
C09672=1060.976,413.204,380.950,175.280,38.404,157.345
C09673=1060.968,412.958,380.995,175.273,38.394,157.342
C09674=1060.958,412.712,381.039,175.266,38.385,157.340
C09675=1060.950,412.466,381.083,175.258,38.376,157.338
C09676=1060.942,412.220,381.128,175.251,38.367,157.335
C09677=1060.933,411.974,381.172,175.244,38.358,157.333
C09678=1060.925,411.728,381.216,175.237,38.349,157.330
C09679=1060.916,411.482,381.261,175.230,38.340,157.328
C09680=1060.908,411.236,381.305,175.221,38.331,157.325
C09681=1060.900,410.990,381.349,175.214,38.322,157.323
C09682=1060.888,410.669,381.407,175.206,38.310,157.320
C09683=1060.877,410.348,381.465,175.196,38.298,157.317
C09684=1060.866,410.027,381.522,175.187,38.287,157.314
C09685=1060.856,409.706,381.579,175.178,38.275,157.311
C09686=1060.847,409.459,381.624,175.171,38.266,157.308
C09687=1060.838,409.214,381.668,175.163,38.258,157.306
C09688=1060.830,408.968,381.712,175.156,38.249,157.303
C09689=1060.823,408.722,381.756,175.149,38.240,157.301
C09690=1060.814,408.476,381.800,175.142,38.231,157.299
C09691=1060.806,408.230,381.843,175.135,38.222,157.296
C09692=1060.798,407.984,381.888,175.129,38.214,157.294
C09693=1060.789,407.738,381.931,175.122,38.205,157.292
C09694=1060.781,407.492,381.975,175.115,38.197,157.290
C09695=1060.773,407.245,382.019,175.108,38.188,157.287
C09696=1060.764,407.000,382.063,175.101,38.179,157.285
C09697=1060.756,406.754,382.106,175.094,38.171,157.283
C09698=1060.748,406.508,382.149,175.087,38.162,157.280
C09699=1060.740,406.262,382.194,175.080,38.154,157.278
C09700=1060.732,406.015,382.237,175.075,38.145,157.276
C09701=1060.724,405.769,382.280,175.068,38.136,157.274
C09702=1060.716,405.523,382.324,175.061,38.128,157.271
C09703=1060.707,405.278,382.368,175.054,38.120,157.269
C09704=1060.700,405.032,382.411,175.047,38.111,157.267
C09705=1060.691,404.786,382.454,175.041,38.103,157.265
C09706=1060.684,404.540,382.498,175.034,38.094,157.263
C09707=1060.675,404.293,382.541,175.027,38.086,157.260
C09708=1060.667,404.047,382.584,175.020,38.078,157.258
C09709=1060.659,403.801,382.627,175.014,38.069,157.256
C09710=1060.650,403.555,382.670,175.008,38.061,157.254
C09711=1060.642,403.309,382.714,175.001,38.053,157.252
C09712=1060.634,403.062,382.756,174.994,38.044,157.249
C09713=1060.626,402.817,382.799,174.987,38.036,157.247
C09714=1060.619,402.573,382.842,174.982,38.028,157.245
C09715=1060.610,402.329,382.884,174.975,38.020,157.243
C09716=1060.603,402.085,382.927,174.968,38.012,157.241
C09717=1060.594,401.841,382.970,174.962,38.004,157.239
C09718=1060.587,401.596,383.012,174.956,37.996,157.237
C09719=1060.578,401.352,383.055,174.949,37.988,157.235
C09720=1060.570,401.109,383.097,174.943,37.980,157.233
C09721=1060.563,400.864,383.139,174.936,37.972,157.230
C09722=1060.555,400.619,383.182,174.930,37.964,157.228
C09723=1060.546,400.372,383.224,174.924,37.956,157.226
C09724=1060.538,400.126,383.267,174.917,37.948,157.224
C09725=1060.530,399.880,383.309,174.911,37.940,157.222
C09726=1060.522,399.634,383.352,174.905,37.932,157.220
C09727=1060.515,399.387,383.395,174.898,37.925,157.218
C09728=1060.507,399.141,383.438,174.892,37.917,157.216
C09729=1060.498,398.895,383.480,174.886,37.908,157.214
C09730=1060.491,398.649,383.522,174.879,37.900,157.212
C09731=1060.483,398.402,383.565,174.873,37.893,157.210
C09732=1060.475,398.157,383.607,174.867,37.885,157.208
C09733=1060.466,397.910,383.650,174.861,37.877,157.206
C09734=1060.459,397.664,383.692,174.855,37.869,157.204
C09735=1060.451,397.417,383.734,174.848,37.861,157.202
C09736=1060.444,397.171,383.776,174.842,37.854,157.200
C09737=1060.436,396.924,383.819,174.836,37.846,157.198
C09738=1060.427,396.679,383.861,174.830,37.838,157.196
C09739=1060.419,396.433,383.903,174.823,37.831,157.194
C09740=1060.411,396.187,383.945,174.818,37.823,157.192
C09741=1060.404,395.941,383.987,174.811,37.815,157.190
C09742=1060.396,395.694,384.029,174.806,37.808,157.188
C09743=1060.388,395.448,384.070,174.799,37.800,157.186
C09744=1060.380,395.201,384.113,174.794,37.793,157.184
C09745=1060.372,394.955,384.155,174.787,37.785,157.182
C09746=1060.365,394.709,384.197,174.781,37.778,157.180
C09747=1060.357,394.463,384.239,174.775,37.770,157.178
C09748=1060.349,394.216,384.281,174.769,37.763,157.176
C09749=1060.342,393.970,384.322,174.763,37.755,157.174
C09750=1060.333,393.724,384.364,174.757,37.748,157.173
C09751=1060.325,393.477,384.406,174.751,37.740,157.171
C09752=1060.318,393.231,384.447,174.745,37.733,157.169
C09753=1060.310,392.985,384.489,174.740,37.725,157.167
C09754=1060.303,392.739,384.531,174.733,37.718,157.165
C09755=1060.295,392.493,384.572,174.728,37.711,157.163
C09756=1060.286,392.246,384.614,174.721,37.703,157.161
C09757=1060.279,391.999,384.655,174.716,37.696,157.159
C09758=1060.272,391.753,384.697,174.709,37.688,157.157
C09759=1060.263,391.507,384.738,174.704,37.681,157.156
C09760=1060.256,391.261,384.780,174.698,37.674,157.154
C09761=1060.249,391.014,384.821,174.692,37.667,157.152
C09762=1060.240,390.767,384.862,174.687,37.659,157.150
C09763=1060.232,390.521,384.904,174.681,37.652,157.148
C09764=1060.225,390.275,384.945,174.675,37.645,157.146
C09765=1060.218,390.028,384.986,174.669,37.638,157.145
C09766=1060.210,389.782,385.027,174.663,37.631,157.143
C09767=1060.202,389.536,385.069,174.657,37.624,157.141
C09768=1060.194,389.290,385.109,174.652,37.617,157.139
C09769=1060.186,389.043,385.150,174.646,37.610,157.137
C09770=1060.179,388.797,385.191,174.640,37.602,157.136
C09771=1060.171,388.551,385.232,174.635,37.595,157.134
C09772=1060.164,388.304,385.273,174.628,37.588,157.132
C09773=1060.156,388.058,385.314,174.623,37.581,157.130
C09774=1060.146,387.757,385.364,174.616,37.573,157.128
C09775=1060.137,387.458,385.414,174.610,37.564,157.126
C09776=1060.127,387.157,385.464,174.602,37.556,157.124
C09777=1060.118,386.857,385.513,174.596,37.547,157.122
C09778=1060.110,386.611,385.554,174.590,37.540,157.120
C09779=1060.103,386.364,385.595,174.584,37.533,157.118
C09780=1060.095,386.118,385.635,174.579,37.526,157.116
C09781=1060.088,385.871,385.676,174.574,37.520,157.115
C09782=1060.080,385.625,385.717,174.567,37.513,157.113
C09783=1060.072,385.379,385.757,174.562,37.506,157.111
C09784=1060.065,385.132,385.798,174.557,37.499,157.110
C09785=1060.057,384.886,385.838,174.552,37.492,157.108
C09786=1060.050,384.639,385.880,174.545,37.485,157.106
C09787=1060.042,384.392,385.920,174.540,37.479,157.104
C09788=1060.034,384.146,385.960,174.535,37.472,157.103
C09789=1060.028,383.900,386.001,174.530,37.465,157.101
C09790=1060.020,383.653,386.041,174.523,37.458,157.099
C09791=1060.013,383.406,386.082,174.518,37.451,157.098
C09792=1060.005,383.159,386.122,174.513,37.445,157.096
C09793=1059.997,382.914,386.162,174.508,37.438,157.094
C09794=1059.990,382.667,386.203,174.501,37.431,157.093
C09795=1059.982,382.420,386.244,174.496,37.425,157.091
C09796=1059.975,382.173,386.283,174.491,37.418,157.089
C09797=1059.968,381.927,386.324,174.486,37.411,157.088
C09798=1059.960,381.681,386.364,174.481,37.405,157.086
C09799=1059.953,381.434,386.404,174.476,37.398,157.084
C09800=1059.946,381.187,386.444,174.469,37.391,157.083
C09801=1059.938,380.941,386.485,174.464,37.384,157.081
C09802=1059.930,380.694,386.525,174.459,37.378,157.079
C09803=1059.924,380.448,386.565,174.454,37.371,157.078
C09804=1059.916,380.201,386.605,174.449,37.365,157.076
C09805=1059.909,379.954,386.645,174.443,37.358,157.074
C09806=1059.901,379.708,386.684,174.437,37.352,157.073
C09807=1059.894,379.461,386.724,174.432,37.346,157.071
C09808=1059.886,379.214,386.764,174.427,37.339,157.070
C09809=1059.879,378.968,386.804,174.422,37.333,157.068
C09810=1059.871,378.721,386.844,174.417,37.326,157.067
C09811=1059.864,378.474,386.883,174.412,37.320,157.065
C09812=1059.856,378.228,386.923,174.407,37.314,157.063
C09813=1059.849,377.981,386.963,174.401,37.307,157.062
C09814=1059.842,377.734,387.003,174.395,37.300,157.060
C09815=1059.834,377.488,387.043,174.390,37.294,157.059
C09816=1059.827,377.241,387.082,174.385,37.288,157.057
C09817=1059.819,376.994,387.122,174.380,37.282,157.056
C09818=1059.812,376.748,387.161,174.375,37.275,157.054
C09819=1059.804,376.501,387.201,174.370,37.269,157.053
C09820=1059.797,376.254,387.240,174.365,37.263,157.051
C09821=1059.790,376.008,387.280,174.360,37.257,157.049
C09822=1059.783,375.761,387.319,174.355,37.250,157.048
C09823=1059.775,375.514,387.359,174.350,37.244,157.046
C09824=1059.768,375.268,387.399,174.344,37.237,157.045
C09825=1059.761,375.021,387.437,174.339,37.231,157.043
C09826=1059.753,374.774,387.477,174.334,37.225,157.042
C09827=1059.747,374.527,387.516,174.329,37.219,157.040
C09828=1059.739,374.280,387.556,174.324,37.213,157.039
C09829=1059.732,374.033,387.595,174.319,37.206,157.037
C09830=1059.723,373.765,387.638,174.313,37.200,157.035
C09831=1059.717,373.496,387.681,174.308,37.193,157.034
C09832=1059.708,373.228,387.724,174.303,37.186,157.032
C09833=1059.700,372.958,387.767,174.297,37.179,157.030
C09834=1059.694,372.712,387.805,174.292,37.173,157.029
C09835=1059.686,372.465,387.845,174.288,37.167,157.028
C09836=1059.679,372.218,387.884,174.283,37.161,157.026
C09837=1059.671,371.971,387.922,174.278,37.155,157.025
C09838=1059.665,371.725,387.961,174.273,37.149,157.023
C09839=1059.657,371.478,388.001,174.268,37.143,157.022
C09840=1059.649,371.231,388.039,174.263,37.137,157.020
C09841=1059.643,370.984,388.078,174.257,37.131,157.019
C09842=1059.635,370.737,388.117,174.253,37.125,157.017
C09843=1059.628,370.490,388.156,174.248,37.119,157.016
C09844=1059.621,370.243,388.194,174.243,37.113,157.014
C09845=1059.613,369.997,388.233,174.238,37.107,157.013
C09846=1059.606,369.750,388.273,174.233,37.101,157.011
C09847=1059.599,369.503,388.311,174.228,37.096,157.010
C09848=1059.591,369.257,388.350,174.223,37.090,157.009
C09849=1059.584,369.010,388.389,174.218,37.083,157.007
C09850=1059.578,368.763,388.427,174.214,37.077,157.006
C09851=1059.570,368.515,388.465,174.209,37.072,157.004
C09852=1059.563,368.268,388.504,174.204,37.066,157.003
C09853=1059.555,368.022,388.542,174.199,37.060,157.002
C09854=1059.549,367.775,388.581,174.194,37.054,157.000
C09855=1059.542,367.528,388.620,174.189,37.048,156.999
C09856=1059.534,367.282,388.658,174.184,37.043,156.997
C09857=1059.527,367.035,388.697,174.179,37.037,156.996
C09858=1059.519,366.787,388.735,174.175,37.031,156.995
C09859=1059.513,366.540,388.774,174.170,37.025,156.993
C09860=1059.506,366.293,388.813,174.165,37.019,156.992
C09861=1059.498,366.047,388.851,174.160,37.013,156.990
C09862=1059.492,365.799,388.889,174.155,37.008,156.989
C09863=1059.484,365.553,388.927,174.150,37.002,156.988
C09864=1059.477,365.306,388.966,174.147,36.996,156.986
C09865=1059.470,365.059,389.004,174.142,36.991,156.985
C09866=1059.463,364.812,389.042,174.137,36.984,156.983
C09867=1059.456,364.566,389.081,174.132,36.979,156.982
C09868=1059.449,364.318,389.119,174.127,36.973,156.981
C09869=1059.443,364.071,389.158,174.123,36.967,156.979
C09870=1059.435,363.824,389.195,174.118,36.962,156.978
C09871=1059.428,363.578,389.233,174.113,36.956,156.977
C09872=1059.421,363.330,389.272,174.108,36.951,156.975
C09873=1059.414,363.083,389.309,174.105,36.945,156.974
C09874=1059.406,362.837,389.347,174.100,36.939,156.973
C09875=1059.400,362.589,389.385,174.095,36.933,156.971
C09876=1059.393,362.342,389.423,174.090,36.928,156.970
C09877=1059.385,362.095,389.461,174.086,36.922,156.969
C09878=1059.379,361.848,389.499,174.081,36.917,156.967
C09879=1059.371,361.601,389.537,174.076,36.911,156.966
C09880=1059.364,361.354,389.575,174.071,36.906,156.965
C09881=1059.357,361.108,389.612,174.068,36.900,156.963
C09882=1059.351,360.861,389.650,174.063,36.895,156.962
C09883=1059.343,360.613,389.688,174.058,36.889,156.961
C09884=1059.336,360.366,389.725,174.053,36.884,156.959
C09885=1059.329,360.119,389.763,174.049,36.878,156.958
C09886=1059.322,359.869,389.802,174.044,36.873,156.957
C09887=1059.315,359.618,389.840,174.039,36.867,156.955
C09888=1059.308,359.367,389.878,174.035,36.862,156.954
C09889=1059.301,359.117,389.917,174.031,36.856,156.953
C09890=1059.294,358.870,389.954,174.026,36.851,156.952
C09891=1059.287,358.623,389.992,174.021,36.845,156.950
C09892=1059.279,358.376,390.029,174.017,36.839,156.949
C09893=1059.273,358.129,390.067,174.012,36.834,156.948
C09894=1059.266,357.882,390.105,174.008,36.829,156.946
C09895=1059.259,357.635,390.142,174.004,36.823,156.945
C09896=1059.252,357.387,390.179,173.999,36.818,156.944
C09897=1059.245,357.140,390.216,173.994,36.813,156.943
C09898=1059.238,356.894,390.254,173.990,36.808,156.941
C09899=1059.231,356.647,390.291,173.986,36.802,156.940
C09900=1059.224,356.399,390.329,173.981,36.797,156.939
C09901=1059.217,356.152,390.365,173.977,36.792,156.938
C09902=1059.210,355.905,390.403,173.972,36.786,156.936
C09903=1059.203,355.658,390.440,173.967,36.781,156.935
C09904=1059.195,355.411,390.478,173.964,36.776,156.934
C09905=1059.189,355.164,390.514,173.959,36.770,156.933
C09906=1059.182,354.917,390.552,173.955,36.765,156.931
C09907=1059.175,354.670,390.589,173.950,36.760,156.930
C09908=1059.168,354.423,390.626,173.945,36.755,156.929
C09909=1059.161,354.175,390.663,173.942,36.749,156.928
C09910=1059.154,353.928,390.700,173.937,36.744,156.926
C09911=1059.148,353.681,390.737,173.933,36.739,156.925
C09912=1059.141,353.434,390.774,173.928,36.733,156.924
C09913=1059.133,353.186,390.811,173.924,36.728,156.923
C09914=1059.127,352.940,390.849,173.920,36.723,156.922
C09915=1059.120,352.692,390.885,173.915,36.718,156.920
C09916=1059.113,352.445,390.922,173.911,36.713,156.919
C09917=1059.106,352.198,390.959,173.907,36.708,156.918
C09918=1059.100,351.951,390.996,173.903,36.703,156.917
C09919=1059.093,351.704,391.033,173.898,36.697,156.915
C09920=1059.086,351.456,391.070,173.894,36.692,156.914
C09921=1059.079,351.209,391.106,173.890,36.687,156.913
C09922=1059.071,350.962,391.143,173.885,36.682,156.912
C09923=1059.065,350.715,391.180,173.881,36.677,156.911
C09924=1059.058,350.467,391.217,173.876,36.672,156.910
C09925=1059.051,350.221,391.253,173.873,36.667,156.908
C09926=1059.044,349.974,391.290,173.868,36.662,156.907
C09927=1059.037,349.726,391.327,173.864,36.657,156.906
C09928=1059.030,349.479,391.363,173.859,36.652,156.905
C09929=1059.023,349.232,391.399,173.856,36.646,156.904
C09930=1059.016,348.984,391.436,173.851,36.641,156.902
C09931=1059.010,348.737,391.472,173.847,36.636,156.901
C09932=1059.003,348.489,391.509,173.843,36.631,156.900
C09933=1058.996,348.243,391.546,173.839,36.626,156.899
C09934=1058.989,347.996,391.583,173.834,36.621,156.898
C09935=1058.983,347.748,391.619,173.830,36.616,156.897
C09936=1058.975,347.501,391.655,173.826,36.611,156.895
C09937=1058.969,347.254,391.692,173.822,36.606,156.894
C09938=1058.961,347.007,391.728,173.817,36.601,156.893
C09939=1058.955,346.760,391.764,173.814,36.596,156.892
C09940=1058.948,346.514,391.801,173.809,36.591,156.891
C09941=1058.942,346.268,391.837,173.805,36.586,156.890
C09942=1058.935,346.021,391.873,173.802,36.581,156.889
C09943=1058.928,345.774,391.908,173.797,36.576,156.887
C09944=1058.921,345.528,391.946,173.793,36.572,156.886
C09945=1058.914,345.281,391.981,173.788,36.567,156.885
C09946=1058.908,345.034,392.018,173.785,36.561,156.884
C09947=1058.901,344.787,392.053,173.780,36.556,156.883
C09948=1058.894,344.539,392.090,173.776,36.552,156.882
C09949=1058.887,344.292,392.126,173.773,36.547,156.881
C09950=1058.881,344.045,392.162,173.768,36.542,156.879
C09951=1058.874,343.797,392.198,173.764,36.537,156.878
C09952=1058.867,343.550,392.234,173.760,36.532,156.877
C09953=1058.861,343.303,392.271,173.756,36.527,156.876
C09954=1058.854,343.056,392.306,173.752,36.523,156.875
C09955=1058.847,342.808,392.342,173.748,36.517,156.874
C09956=1058.840,342.560,392.378,173.744,36.513,156.873
C09957=1058.833,342.314,392.413,173.739,36.508,156.872
C09958=1058.826,342.065,392.450,173.736,36.503,156.871
C09959=1058.819,341.819,392.485,173.732,36.498,156.869
C09960=1058.813,341.571,392.521,173.727,36.494,156.868
C09961=1058.806,341.324,392.557,173.724,36.489,156.867
C09962=1058.799,341.076,392.592,173.719,36.484,156.866
C09963=1058.793,340.829,392.629,173.715,36.479,156.865
C09964=1058.786,340.582,392.664,173.712,36.474,156.864
C09965=1058.779,340.335,392.700,173.707,36.470,156.863
C09966=1058.773,340.087,392.736,173.704,36.465,156.862
C09967=1058.765,339.839,392.771,173.700,36.460,156.861
C09968=1058.758,339.592,392.807,173.695,36.455,156.860
C09969=1058.752,339.345,392.843,173.692,36.451,156.859
C09970=1058.745,339.097,392.878,173.688,36.446,156.858
C09971=1058.738,338.851,392.914,173.683,36.441,156.856
C09972=1058.732,338.603,392.949,173.680,36.436,156.855
C09973=1058.725,338.355,392.985,173.676,36.432,156.854
C09974=1058.718,338.108,393.021,173.671,36.427,156.853
C09975=1058.712,337.861,393.057,173.668,36.422,156.852
C09976=1058.705,337.613,393.092,173.664,36.418,156.851
C09977=1058.698,337.366,393.127,173.661,36.413,156.850
C09978=1058.692,337.118,393.163,173.656,36.408,156.849
C09979=1058.686,336.871,393.198,173.652,36.404,156.848
C09980=1058.678,336.624,393.233,173.649,36.399,156.847
C09981=1058.672,336.377,393.269,173.644,36.395,156.846
C09982=1058.665,336.129,393.304,173.641,36.389,156.845
C09983=1058.658,335.882,393.339,173.637,36.385,156.844
C09984=1058.651,335.634,393.374,173.633,36.380,156.843
C09985=1058.645,335.386,393.410,173.629,36.376,156.842
C09986=1058.638,335.139,393.445,173.625,36.371,156.841
C09987=1058.631,334.891,393.480,173.622,36.367,156.839
C09988=1058.624,334.644,393.516,173.617,36.362,156.838
C09989=1058.618,334.397,393.551,173.613,36.358,156.837
C09990=1058.611,334.149,393.585,173.610,36.353,156.836
C09991=1058.604,333.901,393.620,173.606,36.348,156.835
C09992=1058.598,333.654,393.655,173.602,36.344,156.834
C09993=1058.591,333.407,393.690,173.598,36.339,156.833
C09994=1058.584,333.159,393.726,173.594,36.335,156.832
C09995=1058.577,332.912,393.761,173.591,36.330,156.831
C09996=1058.571,332.665,393.796,173.587,36.326,156.830
//INST
///DATE 2021/06/25 14:47
///ATTR SC,RW,RJ
////FRAME ROBOT
///GROUP1 RB1
NOP
MOVL C00000 V=800.0 PL=0
MOVL C00001 V=800.0 PL=0
MOVL C00002 V=800.0 PL=0
MOVL C00003 V=800.0 PL=0
MOVL C00004 V=800.0 PL=0
MOVL C00005 V=800.0 PL=0
MOVL C00006 V=800.0 PL=0
MOVL C00007 V=800.0 PL=0
MOVL C00008 V=800.0 PL=0
MOVL C00009 V=800.0 PL=0
MOVL C00010 V=800.0 PL=0
MOVL C00011 V=800.0 PL=0
MOVL C00012 V=800.0 PL=0
MOVL C00013 V=800.0 PL=0
MOVL C00014 V=800.0 PL=0
MOVL C00015 V=800.0 PL=0
MOVL C00016 V=800.0 PL=0
MOVL C00017 V=800.0 PL=0
MOVL C00018 V=800.0 PL=0
MOVL C00019 V=800.0 PL=0
MOVL C00020 V=800.0 PL=0
MOVL C00021 V=800.0 PL=0
MOVL C00022 V=800.0 PL=0
MOVL C00023 V=800.0 PL=0
MOVL C00024 V=800.0 PL=0
MOVL C00025 V=800.0 PL=0
MOVL C00026 V=800.0 PL=0
MOVL C00027 V=800.0 PL=0
MOVL C00028 V=800.0 PL=0
MOVL C00029 V=800.0 PL=0
MOVL C00030 V=800.0 PL=0
MOVL C00031 V=800.0 PL=0
MOVL C00032 V=800.0 PL=0
MOVL C00033 V=800.0 PL=0
MOVL C00034 V=800.0 PL=0
MOVL C00035 V=800.0 PL=0
MOVL C00036 V=800.0 PL=0
MOVL C00037 V=800.0 PL=0
MOVL C00038 V=800.0 PL=0
MOVL C00039 V=800.0 PL=0
MOVL C00040 V=800.0 PL=0
MOVL C00041 V=800.0 PL=0
MOVL C00042 V=800.0 PL=0
MOVL C00043 V=800.0 PL=0
MOVL C00044 V=800.0 PL=0
MOVL C00045 V=800.0 PL=0
MOVL C00046 V=800.0 PL=0
MOVL C00047 V=800.0 PL=0
MOVL C00048 V=800.0 PL=0
MOVL C00049 V=800.0 PL=0
MOVL C00050 V=800.0 PL=0
MOVL C00051 V=800.0 PL=0
MOVL C00052 V=800.0 PL=0
MOVL C00053 V=800.0 PL=0
MOVL C00054 V=800.0 PL=0
MOVL C00055 V=800.0 PL=0
MOVL C00056 V=800.0 PL=0
MOVL C00057 V=800.0 PL=0
MOVL C00058 V=800.0 PL=0
MOVL C00059 V=800.0 PL=0
MOVL C00060 V=800.0 PL=0
MOVL C00061 V=800.0 PL=0
MOVL C00062 V=800.0 PL=0
MOVL C00063 V=800.0 PL=0
MOVL C00064 V=800.0 PL=0
MOVL C00065 V=800.0 PL=0
MOVL C00066 V=800.0 PL=0
MOVL C00067 V=800.0 PL=0
MOVL C00068 V=800.0 PL=0
MOVL C00069 V=800.0 PL=0
MOVL C00070 V=800.0 PL=0
MOVL C00071 V=800.0 PL=0
MOVL C00072 V=800.0 PL=0
MOVL C00073 V=800.0 PL=0
MOVL C00074 V=800.0 PL=0
MOVL C00075 V=800.0 PL=0
MOVL C00076 V=800.0 PL=0
MOVL C00077 V=800.0 PL=0
MOVL C00078 V=800.0 PL=0
MOVL C00079 V=800.0 PL=0
MOVL C00080 V=800.0 PL=0
MOVL C00081 V=800.0 PL=0
MOVL C00082 V=800.0 PL=0
MOVL C00083 V=800.0 PL=0
MOVL C00084 V=800.0 PL=0
MOVL C00085 V=800.0 PL=0
MOVL C00086 V=800.0 PL=0
MOVL C00087 V=800.0 PL=0
MOVL C00088 V=800.0 PL=0
MOVL C00089 V=800.0 PL=0
MOVL C00090 V=800.0 PL=0
MOVL C00091 V=800.0 PL=0
MOVL C00092 V=800.0 PL=0
MOVL C00093 V=800.0 PL=0
MOVL C00094 V=800.0 PL=0
MOVL C00095 V=800.0 PL=0
MOVL C00096 V=800.0 PL=0
MOVL C00097 V=800.0 PL=0
MOVL C00098 V=800.0 PL=0
MOVL C00099 V=800.0 PL=0
MOVL C00100 V=800.0 PL=0
MOVL C00101 V=800.0 PL=0
MOVL C00102 V=800.0 PL=0
MOVL C00103 V=800.0 PL=0
MOVL C00104 V=800.0 PL=0
MOVL C00105 V=800.0 PL=0
MOVL C00106 V=800.0 PL=0
MOVL C00107 V=800.0 PL=0
MOVL C00108 V=800.0 PL=0
MOVL C00109 V=800.0 PL=0
MOVL C00110 V=800.0 PL=0
MOVL C00111 V=800.0 PL=0
MOVL C00112 V=800.0 PL=0
MOVL C00113 V=800.0 PL=0
MOVL C00114 V=800.0 PL=0
MOVL C00115 V=800.0 PL=0
MOVL C00116 V=800.0 PL=0
MOVL C00117 V=800.0 PL=0
MOVL C00118 V=800.0 PL=0
MOVL C00119 V=800.0 PL=0
MOVL C00120 V=800.0 PL=0
MOVL C00121 V=800.0 PL=0
MOVL C00122 V=800.0 PL=0
MOVL C00123 V=800.0 PL=0
MOVL C00124 V=800.0 PL=0
MOVL C00125 V=800.0 PL=0
MOVL C00126 V=800.0 PL=0
MOVL C00127 V=800.0 PL=0
MOVL C00128 V=800.0 PL=0
MOVL C00129 V=800.0 PL=0
MOVL C00130 V=800.0 PL=0
MOVL C00131 V=800.0 PL=0
MOVL C00132 V=800.0 PL=0
MOVL C00133 V=800.0 PL=0
MOVL C00134 V=800.0 PL=0
MOVL C00135 V=800.0 PL=0
MOVL C00136 V=800.0 PL=0
MOVL C00137 V=800.0 PL=0
MOVL C00138 V=800.0 PL=0
MOVL C00139 V=800.0 PL=0
MOVL C00140 V=800.0 PL=0
MOVL C00141 V=800.0 PL=0
MOVL C00142 V=800.0 PL=0
MOVL C00143 V=800.0 PL=0
MOVL C00144 V=800.0 PL=0
MOVL C00145 V=800.0 PL=0
MOVL C00146 V=800.0 PL=0
MOVL C00147 V=800.0 PL=0
MOVL C00148 V=800.0 PL=0
MOVL C00149 V=800.0 PL=0
MOVL C00150 V=800.0 PL=0
MOVL C00151 V=800.0 PL=0
MOVL C00152 V=800.0 PL=0
MOVL C00153 V=800.0 PL=0
MOVL C00154 V=800.0 PL=0
MOVL C00155 V=800.0 PL=0
MOVL C00156 V=800.0 PL=0
MOVL C00157 V=800.0 PL=0
MOVL C00158 V=800.0 PL=0
MOVL C00159 V=800.0 PL=0
MOVL C00160 V=800.0 PL=0
MOVL C00161 V=800.0 PL=0
MOVL C00162 V=800.0 PL=0
MOVL C00163 V=800.0 PL=0
MOVL C00164 V=800.0 PL=0
MOVL C00165 V=800.0 PL=0
MOVL C00166 V=800.0 PL=0
MOVL C00167 V=800.0 PL=0
MOVL C00168 V=800.0 PL=0
MOVL C00169 V=800.0 PL=0
MOVL C00170 V=800.0 PL=0
MOVL C00171 V=800.0 PL=0
MOVL C00172 V=800.0 PL=0
MOVL C00173 V=800.0 PL=0
MOVL C00174 V=800.0 PL=0
MOVL C00175 V=800.0 PL=0
MOVL C00176 V=800.0 PL=0
MOVL C00177 V=800.0 PL=0
MOVL C00178 V=800.0 PL=0
MOVL C00179 V=800.0 PL=0
MOVL C00180 V=800.0 PL=0
MOVL C00181 V=800.0 PL=0
MOVL C00182 V=800.0 PL=0
MOVL C00183 V=800.0 PL=0
MOVL C00184 V=800.0 PL=0
MOVL C00185 V=800.0 PL=0
MOVL C00186 V=800.0 PL=0
MOVL C00187 V=800.0 PL=0
MOVL C00188 V=800.0 PL=0
MOVL C00189 V=800.0 PL=0
MOVL C00190 V=800.0 PL=0
MOVL C00191 V=800.0 PL=0
MOVL C00192 V=800.0 PL=0
MOVL C00193 V=800.0 PL=0
MOVL C00194 V=800.0 PL=0
MOVL C00195 V=800.0 PL=0
MOVL C00196 V=800.0 PL=0
MOVL C00197 V=800.0 PL=0
MOVL C00198 V=800.0 PL=0
MOVL C00199 V=800.0 PL=0
MOVL C00200 V=800.0 PL=0
MOVL C00201 V=800.0 PL=0
MOVL C00202 V=800.0 PL=0
MOVL C00203 V=800.0 PL=0
MOVL C00204 V=800.0 PL=0
MOVL C00205 V=800.0 PL=0
MOVL C00206 V=800.0 PL=0
MOVL C00207 V=800.0 PL=0
MOVL C00208 V=800.0 PL=0
MOVL C00209 V=800.0 PL=0
MOVL C00210 V=800.0 PL=0
MOVL C00211 V=800.0 PL=0
MOVL C00212 V=800.0 PL=0
MOVL C00213 V=800.0 PL=0
MOVL C00214 V=800.0 PL=0
MOVL C00215 V=800.0 PL=0
MOVL C00216 V=800.0 PL=0
MOVL C00217 V=800.0 PL=0
MOVL C00218 V=800.0 PL=0
MOVL C00219 V=800.0 PL=0
MOVL C00220 V=800.0 PL=0
MOVL C00221 V=800.0 PL=0
MOVL C00222 V=800.0 PL=0
MOVL C00223 V=800.0 PL=0
MOVL C00224 V=800.0 PL=0
MOVL C00225 V=800.0 PL=0
MOVL C00226 V=800.0 PL=0
MOVL C00227 V=800.0 PL=0
MOVL C00228 V=800.0 PL=0
MOVL C00229 V=800.0 PL=0
MOVL C00230 V=800.0 PL=0
MOVL C00231 V=800.0 PL=0
MOVL C00232 V=800.0 PL=0
MOVL C00233 V=800.0 PL=0
MOVL C00234 V=800.0 PL=0
MOVL C00235 V=800.0 PL=0
MOVL C00236 V=800.0 PL=0
MOVL C00237 V=800.0 PL=0
MOVL C00238 V=800.0 PL=0
MOVL C00239 V=800.0 PL=0
MOVL C00240 V=800.0 PL=0
MOVL C00241 V=800.0 PL=0
MOVL C00242 V=800.0 PL=0
MOVL C00243 V=800.0 PL=0
MOVL C00244 V=800.0 PL=0
MOVL C00245 V=800.0 PL=0
MOVL C00246 V=800.0 PL=0
MOVL C00247 V=800.0 PL=0
MOVL C00248 V=800.0 PL=0
MOVL C00249 V=800.0 PL=0
MOVL C00250 V=800.0 PL=0
MOVL C00251 V=800.0 PL=0
MOVL C00252 V=800.0 PL=0
MOVL C00253 V=800.0 PL=0
MOVL C00254 V=800.0 PL=0
MOVL C00255 V=800.0 PL=0
MOVL C00256 V=800.0 PL=0
MOVL C00257 V=800.0 PL=0
MOVL C00258 V=800.0 PL=0
MOVL C00259 V=800.0 PL=0
MOVL C00260 V=800.0 PL=0
MOVL C00261 V=800.0 PL=0
MOVL C00262 V=800.0 PL=0
MOVL C00263 V=800.0 PL=0
MOVL C00264 V=800.0 PL=0
MOVL C00265 V=800.0 PL=0
MOVL C00266 V=800.0 PL=0
MOVL C00267 V=800.0 PL=0
MOVL C00268 V=800.0 PL=0
MOVL C00269 V=800.0 PL=0
MOVL C00270 V=800.0 PL=0
MOVL C00271 V=800.0 PL=0
MOVL C00272 V=800.0 PL=0
MOVL C00273 V=800.0 PL=0
MOVL C00274 V=800.0 PL=0
MOVL C00275 V=800.0 PL=0
MOVL C00276 V=800.0 PL=0
MOVL C00277 V=800.0 PL=0
MOVL C00278 V=800.0 PL=0
MOVL C00279 V=800.0 PL=0
MOVL C00280 V=800.0 PL=0
MOVL C00281 V=800.0 PL=0
MOVL C00282 V=800.0 PL=0
MOVL C00283 V=800.0 PL=0
MOVL C00284 V=800.0 PL=0
MOVL C00285 V=800.0 PL=0
MOVL C00286 V=800.0 PL=0
MOVL C00287 V=800.0 PL=0
MOVL C00288 V=800.0 PL=0
MOVL C00289 V=800.0 PL=0
MOVL C00290 V=800.0 PL=0
MOVL C00291 V=800.0 PL=0
MOVL C00292 V=800.0 PL=0
MOVL C00293 V=800.0 PL=0
MOVL C00294 V=800.0 PL=0
MOVL C00295 V=800.0 PL=0
MOVL C00296 V=800.0 PL=0
MOVL C00297 V=800.0 PL=0
MOVL C00298 V=800.0 PL=0
MOVL C00299 V=800.0 PL=0
MOVL C00300 V=800.0 PL=0
MOVL C00301 V=800.0 PL=0
MOVL C00302 V=800.0 PL=0
MOVL C00303 V=800.0 PL=0
MOVL C00304 V=800.0 PL=0
MOVL C00305 V=800.0 PL=0
MOVL C00306 V=800.0 PL=0
MOVL C00307 V=800.0 PL=0
MOVL C00308 V=800.0 PL=0
MOVL C00309 V=800.0 PL=0
MOVL C00310 V=800.0 PL=0
MOVL C00311 V=800.0 PL=0
MOVL C00312 V=800.0 PL=0
MOVL C00313 V=800.0 PL=0
MOVL C00314 V=800.0 PL=0
MOVL C00315 V=800.0 PL=0
MOVL C00316 V=800.0 PL=0
MOVL C00317 V=800.0 PL=0
MOVL C00318 V=800.0 PL=0
MOVL C00319 V=800.0 PL=0
MOVL C00320 V=800.0 PL=0
MOVL C00321 V=800.0 PL=0
MOVL C00322 V=800.0 PL=0
MOVL C00323 V=800.0 PL=0
MOVL C00324 V=800.0 PL=0
MOVL C00325 V=800.0 PL=0
MOVL C00326 V=800.0 PL=0
MOVL C00327 V=800.0 PL=0
MOVL C00328 V=800.0 PL=0
MOVL C00329 V=800.0 PL=0
MOVL C00330 V=800.0 PL=0
MOVL C00331 V=800.0 PL=0
MOVL C00332 V=800.0 PL=0
MOVL C00333 V=800.0 PL=0
MOVL C00334 V=800.0 PL=0
MOVL C00335 V=800.0 PL=0
MOVL C00336 V=800.0 PL=0
MOVL C00337 V=800.0 PL=0
MOVL C00338 V=800.0 PL=0
MOVL C00339 V=800.0 PL=0
MOVL C00340 V=800.0 PL=0
MOVL C00341 V=800.0 PL=0
MOVL C00342 V=800.0 PL=0
MOVL C00343 V=800.0 PL=0
MOVL C00344 V=800.0 PL=0
MOVL C00345 V=800.0 PL=0
MOVL C00346 V=800.0 PL=0
MOVL C00347 V=800.0 PL=0
MOVL C00348 V=800.0 PL=0
MOVL C00349 V=800.0 PL=0
MOVL C00350 V=800.0 PL=0
MOVL C00351 V=800.0 PL=0
MOVL C00352 V=800.0 PL=0
MOVL C00353 V=800.0 PL=0
MOVL C00354 V=800.0 PL=0
MOVL C00355 V=800.0 PL=0
MOVL C00356 V=800.0 PL=0
MOVL C00357 V=800.0 PL=0
MOVL C00358 V=800.0 PL=0
MOVL C00359 V=800.0 PL=0
MOVL C00360 V=800.0 PL=0
MOVL C00361 V=800.0 PL=0
MOVL C00362 V=800.0 PL=0
MOVL C00363 V=800.0 PL=0
MOVL C00364 V=800.0 PL=0
MOVL C00365 V=800.0 PL=0
MOVL C00366 V=800.0 PL=0
MOVL C00367 V=800.0 PL=0
MOVL C00368 V=800.0 PL=0
MOVL C00369 V=800.0 PL=0
MOVL C00370 V=800.0 PL=0
MOVL C00371 V=800.0 PL=0
MOVL C00372 V=800.0 PL=0
MOVL C00373 V=800.0 PL=0
MOVL C00374 V=800.0 PL=0
MOVL C00375 V=800.0 PL=0
MOVL C00376 V=800.0 PL=0
MOVL C00377 V=800.0 PL=0
MOVL C00378 V=800.0 PL=0
MOVL C00379 V=800.0 PL=0
MOVL C00380 V=800.0 PL=0
MOVL C00381 V=800.0 PL=0
MOVL C00382 V=800.0 PL=0
MOVL C00383 V=800.0 PL=0
MOVL C00384 V=800.0 PL=0
MOVL C00385 V=800.0 PL=0
MOVL C00386 V=800.0 PL=0
MOVL C00387 V=800.0 PL=0
MOVL C00388 V=800.0 PL=0
MOVL C00389 V=800.0 PL=0
MOVL C00390 V=800.0 PL=0
MOVL C00391 V=800.0 PL=0
MOVL C00392 V=800.0 PL=0
MOVL C00393 V=800.0 PL=0
MOVL C00394 V=800.0 PL=0
MOVL C00395 V=800.0 PL=0
MOVL C00396 V=800.0 PL=0
MOVL C00397 V=800.0 PL=0
MOVL C00398 V=800.0 PL=0
MOVL C00399 V=800.0 PL=0
MOVL C00400 V=800.0 PL=0
MOVL C00401 V=800.0 PL=0
MOVL C00402 V=800.0 PL=0
MOVL C00403 V=800.0 PL=0
MOVL C00404 V=800.0 PL=0
MOVL C00405 V=800.0 PL=0
MOVL C00406 V=800.0 PL=0
MOVL C00407 V=800.0 PL=0
MOVL C00408 V=800.0 PL=0
MOVL C00409 V=800.0 PL=0
MOVL C00410 V=800.0 PL=0
MOVL C00411 V=800.0 PL=0
MOVL C00412 V=800.0 PL=0
MOVL C00413 V=800.0 PL=0
MOVL C00414 V=800.0 PL=0
MOVL C00415 V=800.0 PL=0
MOVL C00416 V=800.0 PL=0
MOVL C00417 V=800.0 PL=0
MOVL C00418 V=800.0 PL=0
MOVL C00419 V=800.0 PL=0
MOVL C00420 V=800.0 PL=0
MOVL C00421 V=800.0 PL=0
MOVL C00422 V=800.0 PL=0
MOVL C00423 V=800.0 PL=0
MOVL C00424 V=800.0 PL=0
MOVL C00425 V=800.0 PL=0
MOVL C00426 V=800.0 PL=0
MOVL C00427 V=800.0 PL=0
MOVL C00428 V=800.0 PL=0
MOVL C00429 V=800.0 PL=0
MOVL C00430 V=800.0 PL=0
MOVL C00431 V=800.0 PL=0
MOVL C00432 V=800.0 PL=0
MOVL C00433 V=800.0 PL=0
MOVL C00434 V=800.0 PL=0
MOVL C00435 V=800.0 PL=0
MOVL C00436 V=800.0 PL=0
MOVL C00437 V=800.0 PL=0
MOVL C00438 V=800.0 PL=0
MOVL C00439 V=800.0 PL=0
MOVL C00440 V=800.0 PL=0
MOVL C00441 V=800.0 PL=0
MOVL C00442 V=800.0 PL=0
MOVL C00443 V=800.0 PL=0
MOVL C00444 V=800.0 PL=0
MOVL C00445 V=800.0 PL=0
MOVL C00446 V=800.0 PL=0
MOVL C00447 V=800.0 PL=0
MOVL C00448 V=800.0 PL=0
MOVL C00449 V=800.0 PL=0
MOVL C00450 V=800.0 PL=0
MOVL C00451 V=800.0 PL=0
MOVL C00452 V=800.0 PL=0
MOVL C00453 V=800.0 PL=0
MOVL C00454 V=800.0 PL=0
MOVL C00455 V=800.0 PL=0
MOVL C00456 V=800.0 PL=0
MOVL C00457 V=800.0 PL=0
MOVL C00458 V=800.0 PL=0
MOVL C00459 V=800.0 PL=0
MOVL C00460 V=800.0 PL=0
MOVL C00461 V=800.0 PL=0
MOVL C00462 V=800.0 PL=0
MOVL C00463 V=800.0 PL=0
MOVL C00464 V=800.0 PL=0
MOVL C00465 V=800.0 PL=0
MOVL C00466 V=800.0 PL=0
MOVL C00467 V=800.0 PL=0
MOVL C00468 V=800.0 PL=0
MOVL C00469 V=800.0 PL=0
MOVL C00470 V=800.0 PL=0
MOVL C00471 V=800.0 PL=0
MOVL C00472 V=800.0 PL=0
MOVL C00473 V=800.0 PL=0
MOVL C00474 V=800.0 PL=0
MOVL C00475 V=800.0 PL=0
MOVL C00476 V=800.0 PL=0
MOVL C00477 V=800.0 PL=0
MOVL C00478 V=800.0 PL=0
MOVL C00479 V=800.0 PL=0
MOVL C00480 V=800.0 PL=0
MOVL C00481 V=800.0 PL=0
MOVL C00482 V=800.0 PL=0
MOVL C00483 V=800.0 PL=0
MOVL C00484 V=800.0 PL=0
MOVL C00485 V=800.0 PL=0
MOVL C00486 V=800.0 PL=0
MOVL C00487 V=800.0 PL=0
MOVL C00488 V=800.0 PL=0
MOVL C00489 V=800.0 PL=0
MOVL C00490 V=800.0 PL=0
MOVL C00491 V=800.0 PL=0
MOVL C00492 V=800.0 PL=0
MOVL C00493 V=800.0 PL=0
MOVL C00494 V=800.0 PL=0
MOVL C00495 V=800.0 PL=0
MOVL C00496 V=800.0 PL=0
MOVL C00497 V=800.0 PL=0
MOVL C00498 V=800.0 PL=0
MOVL C00499 V=800.0 PL=0
MOVL C00500 V=800.0 PL=0
MOVL C00501 V=800.0 PL=0
MOVL C00502 V=800.0 PL=0
MOVL C00503 V=800.0 PL=0
MOVL C00504 V=800.0 PL=0
MOVL C00505 V=800.0 PL=0
MOVL C00506 V=800.0 PL=0
MOVL C00507 V=800.0 PL=0
MOVL C00508 V=800.0 PL=0
MOVL C00509 V=800.0 PL=0
MOVL C00510 V=800.0 PL=0
MOVL C00511 V=800.0 PL=0
MOVL C00512 V=800.0 PL=0
MOVL C00513 V=800.0 PL=0
MOVL C00514 V=800.0 PL=0
MOVL C00515 V=800.0 PL=0
MOVL C00516 V=800.0 PL=0
MOVL C00517 V=800.0 PL=0
MOVL C00518 V=800.0 PL=0
MOVL C00519 V=800.0 PL=0
MOVL C00520 V=800.0 PL=0
MOVL C00521 V=800.0 PL=0
MOVL C00522 V=800.0 PL=0
MOVL C00523 V=800.0 PL=0
MOVL C00524 V=800.0 PL=0
MOVL C00525 V=800.0 PL=0
MOVL C00526 V=800.0 PL=0
MOVL C00527 V=800.0 PL=0
MOVL C00528 V=800.0 PL=0
MOVL C00529 V=800.0 PL=0
MOVL C00530 V=800.0 PL=0
MOVL C00531 V=800.0 PL=0
MOVL C00532 V=800.0 PL=0
MOVL C00533 V=800.0 PL=0
MOVL C00534 V=800.0 PL=0
MOVL C00535 V=800.0 PL=0
MOVL C00536 V=800.0 PL=0
MOVL C00537 V=800.0 PL=0
MOVL C00538 V=800.0 PL=0
MOVL C00539 V=800.0 PL=0
MOVL C00540 V=800.0 PL=0
MOVL C00541 V=800.0 PL=0
MOVL C00542 V=800.0 PL=0
MOVL C00543 V=800.0 PL=0
MOVL C00544 V=800.0 PL=0
MOVL C00545 V=800.0 PL=0
MOVL C00546 V=800.0 PL=0
MOVL C00547 V=800.0 PL=0
MOVL C00548 V=800.0 PL=0
MOVL C00549 V=800.0 PL=0
MOVL C00550 V=800.0 PL=0
MOVL C00551 V=800.0 PL=0
MOVL C00552 V=800.0 PL=0
MOVL C00553 V=800.0 PL=0
MOVL C00554 V=800.0 PL=0
MOVL C00555 V=800.0 PL=0
MOVL C00556 V=800.0 PL=0
MOVL C00557 V=800.0 PL=0
MOVL C00558 V=800.0 PL=0
MOVL C00559 V=800.0 PL=0
MOVL C00560 V=800.0 PL=0
MOVL C00561 V=800.0 PL=0
MOVL C00562 V=800.0 PL=0
MOVL C00563 V=800.0 PL=0
MOVL C00564 V=800.0 PL=0
MOVL C00565 V=800.0 PL=0
MOVL C00566 V=800.0 PL=0
MOVL C00567 V=800.0 PL=0
MOVL C00568 V=800.0 PL=0
MOVL C00569 V=800.0 PL=0
MOVL C00570 V=800.0 PL=0
MOVL C00571 V=800.0 PL=0
MOVL C00572 V=800.0 PL=0
MOVL C00573 V=800.0 PL=0
MOVL C00574 V=800.0 PL=0
MOVL C00575 V=800.0 PL=0
MOVL C00576 V=800.0 PL=0
MOVL C00577 V=800.0 PL=0
MOVL C00578 V=800.0 PL=0
MOVL C00579 V=800.0 PL=0
MOVL C00580 V=800.0 PL=0
MOVL C00581 V=800.0 PL=0
MOVL C00582 V=800.0 PL=0
MOVL C00583 V=800.0 PL=0
MOVL C00584 V=800.0 PL=0
MOVL C00585 V=800.0 PL=0
MOVL C00586 V=800.0 PL=0
MOVL C00587 V=800.0 PL=0
MOVL C00588 V=800.0 PL=0
MOVL C00589 V=800.0 PL=0
MOVL C00590 V=800.0 PL=0
MOVL C00591 V=800.0 PL=0
MOVL C00592 V=800.0 PL=0
MOVL C00593 V=800.0 PL=0
MOVL C00594 V=800.0 PL=0
MOVL C00595 V=800.0 PL=0
MOVL C00596 V=800.0 PL=0
MOVL C00597 V=800.0 PL=0
MOVL C00598 V=800.0 PL=0
MOVL C00599 V=800.0 PL=0
MOVL C00600 V=800.0 PL=0
MOVL C00601 V=800.0 PL=0
MOVL C00602 V=800.0 PL=0
MOVL C00603 V=800.0 PL=0
MOVL C00604 V=800.0 PL=0
MOVL C00605 V=800.0 PL=0
MOVL C00606 V=800.0 PL=0
MOVL C00607 V=800.0 PL=0
MOVL C00608 V=800.0 PL=0
MOVL C00609 V=800.0 PL=0
MOVL C00610 V=800.0 PL=0
MOVL C00611 V=800.0 PL=0
MOVL C00612 V=800.0 PL=0
MOVL C00613 V=800.0 PL=0
MOVL C00614 V=800.0 PL=0
MOVL C00615 V=800.0 PL=0
MOVL C00616 V=800.0 PL=0
MOVL C00617 V=800.0 PL=0
MOVL C00618 V=800.0 PL=0
MOVL C00619 V=800.0 PL=0
MOVL C00620 V=800.0 PL=0
MOVL C00621 V=800.0 PL=0
MOVL C00622 V=800.0 PL=0
MOVL C00623 V=800.0 PL=0
MOVL C00624 V=800.0 PL=0
MOVL C00625 V=800.0 PL=0
MOVL C00626 V=800.0 PL=0
MOVL C00627 V=800.0 PL=0
MOVL C00628 V=800.0 PL=0
MOVL C00629 V=800.0 PL=0
MOVL C00630 V=800.0 PL=0
MOVL C00631 V=800.0 PL=0
MOVL C00632 V=800.0 PL=0
MOVL C00633 V=800.0 PL=0
MOVL C00634 V=800.0 PL=0
MOVL C00635 V=800.0 PL=0
MOVL C00636 V=800.0 PL=0
MOVL C00637 V=800.0 PL=0
MOVL C00638 V=800.0 PL=0
MOVL C00639 V=800.0 PL=0
MOVL C00640 V=800.0 PL=0
MOVL C00641 V=800.0 PL=0
MOVL C00642 V=800.0 PL=0
MOVL C00643 V=800.0 PL=0
MOVL C00644 V=800.0 PL=0
MOVL C00645 V=800.0 PL=0
MOVL C00646 V=800.0 PL=0
MOVL C00647 V=800.0 PL=0
MOVL C00648 V=800.0 PL=0
MOVL C00649 V=800.0 PL=0
MOVL C00650 V=800.0 PL=0
MOVL C00651 V=800.0 PL=0
MOVL C00652 V=800.0 PL=0
MOVL C00653 V=800.0 PL=0
MOVL C00654 V=800.0 PL=0
MOVL C00655 V=800.0 PL=0
MOVL C00656 V=800.0 PL=0
MOVL C00657 V=800.0 PL=0
MOVL C00658 V=800.0 PL=0
MOVL C00659 V=800.0 PL=0
MOVL C00660 V=800.0 PL=0
MOVL C00661 V=800.0 PL=0
MOVL C00662 V=800.0 PL=0
MOVL C00663 V=800.0 PL=0
MOVL C00664 V=800.0 PL=0
MOVL C00665 V=800.0 PL=0
MOVL C00666 V=800.0 PL=0
MOVL C00667 V=800.0 PL=0
MOVL C00668 V=800.0 PL=0
MOVL C00669 V=800.0 PL=0
MOVL C00670 V=800.0 PL=0
MOVL C00671 V=800.0 PL=0
MOVL C00672 V=800.0 PL=0
MOVL C00673 V=800.0 PL=0
MOVL C00674 V=800.0 PL=0
MOVL C00675 V=800.0 PL=0
MOVL C00676 V=800.0 PL=0
MOVL C00677 V=800.0 PL=0
MOVL C00678 V=800.0 PL=0
MOVL C00679 V=800.0 PL=0
MOVL C00680 V=800.0 PL=0
MOVL C00681 V=800.0 PL=0
MOVL C00682 V=800.0 PL=0
MOVL C00683 V=800.0 PL=0
MOVL C00684 V=800.0 PL=0
MOVL C00685 V=800.0 PL=0
MOVL C00686 V=800.0 PL=0
MOVL C00687 V=800.0 PL=0
MOVL C00688 V=800.0 PL=0
MOVL C00689 V=800.0 PL=0
MOVL C00690 V=800.0 PL=0
MOVL C00691 V=800.0 PL=0
MOVL C00692 V=800.0 PL=0
MOVL C00693 V=800.0 PL=0
MOVL C00694 V=800.0 PL=0
MOVL C00695 V=800.0 PL=0
MOVL C00696 V=800.0 PL=0
MOVL C00697 V=800.0 PL=0
MOVL C00698 V=800.0 PL=0
MOVL C00699 V=800.0 PL=0
MOVL C00700 V=800.0 PL=0
MOVL C00701 V=800.0 PL=0
MOVL C00702 V=800.0 PL=0
MOVL C00703 V=800.0 PL=0
MOVL C00704 V=800.0 PL=0
MOVL C00705 V=800.0 PL=0
MOVL C00706 V=800.0 PL=0
MOVL C00707 V=800.0 PL=0
MOVL C00708 V=800.0 PL=0
MOVL C00709 V=800.0 PL=0
MOVL C00710 V=800.0 PL=0
MOVL C00711 V=800.0 PL=0
MOVL C00712 V=800.0 PL=0
MOVL C00713 V=800.0 PL=0
MOVL C00714 V=800.0 PL=0
MOVL C00715 V=800.0 PL=0
MOVL C00716 V=800.0 PL=0
MOVL C00717 V=800.0 PL=0
MOVL C00718 V=800.0 PL=0
MOVL C00719 V=800.0 PL=0
MOVL C00720 V=800.0 PL=0
MOVL C00721 V=800.0 PL=0
MOVL C00722 V=800.0 PL=0
MOVL C00723 V=800.0 PL=0
MOVL C00724 V=800.0 PL=0
MOVL C00725 V=800.0 PL=0
MOVL C00726 V=800.0 PL=0
MOVL C00727 V=800.0 PL=0
MOVL C00728 V=800.0 PL=0
MOVL C00729 V=800.0 PL=0
MOVL C00730 V=800.0 PL=0
MOVL C00731 V=800.0 PL=0
MOVL C00732 V=800.0 PL=0
MOVL C00733 V=800.0 PL=0
MOVL C00734 V=800.0 PL=0
MOVL C00735 V=800.0 PL=0
MOVL C00736 V=800.0 PL=0
MOVL C00737 V=800.0 PL=0
MOVL C00738 V=800.0 PL=0
MOVL C00739 V=800.0 PL=0
MOVL C00740 V=800.0 PL=0
MOVL C00741 V=800.0 PL=0
MOVL C00742 V=800.0 PL=0
MOVL C00743 V=800.0 PL=0
MOVL C00744 V=800.0 PL=0
MOVL C00745 V=800.0 PL=0
MOVL C00746 V=800.0 PL=0
MOVL C00747 V=800.0 PL=0
MOVL C00748 V=800.0 PL=0
MOVL C00749 V=800.0 PL=0
MOVL C00750 V=800.0 PL=0
MOVL C00751 V=800.0 PL=0
MOVL C00752 V=800.0 PL=0
MOVL C00753 V=800.0 PL=0
MOVL C00754 V=800.0 PL=0
MOVL C00755 V=800.0 PL=0
MOVL C00756 V=800.0 PL=0
MOVL C00757 V=800.0 PL=0
MOVL C00758 V=800.0 PL=0
MOVL C00759 V=800.0 PL=0
MOVL C00760 V=800.0 PL=0
MOVL C00761 V=800.0 PL=0
MOVL C00762 V=800.0 PL=0
MOVL C00763 V=800.0 PL=0
MOVL C00764 V=800.0 PL=0
MOVL C00765 V=800.0 PL=0
MOVL C00766 V=800.0 PL=0
MOVL C00767 V=800.0 PL=0
MOVL C00768 V=800.0 PL=0
MOVL C00769 V=800.0 PL=0
MOVL C00770 V=800.0 PL=0
MOVL C00771 V=800.0 PL=0
MOVL C00772 V=800.0 PL=0
MOVL C00773 V=800.0 PL=0
MOVL C00774 V=800.0 PL=0
MOVL C00775 V=800.0 PL=0
MOVL C00776 V=800.0 PL=0
MOVL C00777 V=800.0 PL=0
MOVL C00778 V=800.0 PL=0
MOVL C00779 V=800.0 PL=0
MOVL C00780 V=800.0 PL=0
MOVL C00781 V=800.0 PL=0
MOVL C00782 V=800.0 PL=0
MOVL C00783 V=800.0 PL=0
MOVL C00784 V=800.0 PL=0
MOVL C00785 V=800.0 PL=0
MOVL C00786 V=800.0 PL=0
MOVL C00787 V=800.0 PL=0
MOVL C00788 V=800.0 PL=0
MOVL C00789 V=800.0 PL=0
MOVL C00790 V=800.0 PL=0
MOVL C00791 V=800.0 PL=0
MOVL C00792 V=800.0 PL=0
MOVL C00793 V=800.0 PL=0
MOVL C00794 V=800.0 PL=0
MOVL C00795 V=800.0 PL=0
MOVL C00796 V=800.0 PL=0
MOVL C00797 V=800.0 PL=0
MOVL C00798 V=800.0 PL=0
MOVL C00799 V=800.0 PL=0
MOVL C00800 V=800.0 PL=0
MOVL C00801 V=800.0 PL=0
MOVL C00802 V=800.0 PL=0
MOVL C00803 V=800.0 PL=0
MOVL C00804 V=800.0 PL=0
MOVL C00805 V=800.0 PL=0
MOVL C00806 V=800.0 PL=0
MOVL C00807 V=800.0 PL=0
MOVL C00808 V=800.0 PL=0
MOVL C00809 V=800.0 PL=0
MOVL C00810 V=800.0 PL=0
MOVL C00811 V=800.0 PL=0
MOVL C00812 V=800.0 PL=0
MOVL C00813 V=800.0 PL=0
MOVL C00814 V=800.0 PL=0
MOVL C00815 V=800.0 PL=0
MOVL C00816 V=800.0 PL=0
MOVL C00817 V=800.0 PL=0
MOVL C00818 V=800.0 PL=0
MOVL C00819 V=800.0 PL=0
MOVL C00820 V=800.0 PL=0
MOVL C00821 V=800.0 PL=0
MOVL C00822 V=800.0 PL=0
MOVL C00823 V=800.0 PL=0
MOVL C00824 V=800.0 PL=0
MOVL C00825 V=800.0 PL=0
MOVL C00826 V=800.0 PL=0
MOVL C00827 V=800.0 PL=0
MOVL C00828 V=800.0 PL=0
MOVL C00829 V=800.0 PL=0
MOVL C00830 V=800.0 PL=0
MOVL C00831 V=800.0 PL=0
MOVL C00832 V=800.0 PL=0
MOVL C00833 V=800.0 PL=0
MOVL C00834 V=800.0 PL=0
MOVL C00835 V=800.0 PL=0
MOVL C00836 V=800.0 PL=0
MOVL C00837 V=800.0 PL=0
MOVL C00838 V=800.0 PL=0
MOVL C00839 V=800.0 PL=0
MOVL C00840 V=800.0 PL=0
MOVL C00841 V=800.0 PL=0
MOVL C00842 V=800.0 PL=0
MOVL C00843 V=800.0 PL=0
MOVL C00844 V=800.0 PL=0
MOVL C00845 V=800.0 PL=0
MOVL C00846 V=800.0 PL=0
MOVL C00847 V=800.0 PL=0
MOVL C00848 V=800.0 PL=0
MOVL C00849 V=800.0 PL=0
MOVL C00850 V=800.0 PL=0
MOVL C00851 V=800.0 PL=0
MOVL C00852 V=800.0 PL=0
MOVL C00853 V=800.0 PL=0
MOVL C00854 V=800.0 PL=0
MOVL C00855 V=800.0 PL=0
MOVL C00856 V=800.0 PL=0
MOVL C00857 V=800.0 PL=0
MOVL C00858 V=800.0 PL=0
MOVL C00859 V=800.0 PL=0
MOVL C00860 V=800.0 PL=0
MOVL C00861 V=800.0 PL=0
MOVL C00862 V=800.0 PL=0
MOVL C00863 V=800.0 PL=0
MOVL C00864 V=800.0 PL=0
MOVL C00865 V=800.0 PL=0
MOVL C00866 V=800.0 PL=0
MOVL C00867 V=800.0 PL=0
MOVL C00868 V=800.0 PL=0
MOVL C00869 V=800.0 PL=0
MOVL C00870 V=800.0 PL=0
MOVL C00871 V=800.0 PL=0
MOVL C00872 V=800.0 PL=0
MOVL C00873 V=800.0 PL=0
MOVL C00874 V=800.0 PL=0
MOVL C00875 V=800.0 PL=0
MOVL C00876 V=800.0 PL=0
MOVL C00877 V=800.0 PL=0
MOVL C00878 V=800.0 PL=0
MOVL C00879 V=800.0 PL=0
MOVL C00880 V=800.0 PL=0
MOVL C00881 V=800.0 PL=0
MOVL C00882 V=800.0 PL=0
MOVL C00883 V=800.0 PL=0
MOVL C00884 V=800.0 PL=0
MOVL C00885 V=800.0 PL=0
MOVL C00886 V=800.0 PL=0
MOVL C00887 V=800.0 PL=0
MOVL C00888 V=800.0 PL=0
MOVL C00889 V=800.0 PL=0
MOVL C00890 V=800.0 PL=0
MOVL C00891 V=800.0 PL=0
MOVL C00892 V=800.0 PL=0
MOVL C00893 V=800.0 PL=0
MOVL C00894 V=800.0 PL=0
MOVL C00895 V=800.0 PL=0
MOVL C00896 V=800.0 PL=0
MOVL C00897 V=800.0 PL=0
MOVL C00898 V=800.0 PL=0
MOVL C00899 V=800.0 PL=0
MOVL C00900 V=800.0 PL=0
MOVL C00901 V=800.0 PL=0
MOVL C00902 V=800.0 PL=0
MOVL C00903 V=800.0 PL=0
MOVL C00904 V=800.0 PL=0
MOVL C00905 V=800.0 PL=0
MOVL C00906 V=800.0 PL=0
MOVL C00907 V=800.0 PL=0
MOVL C00908 V=800.0 PL=0
MOVL C00909 V=800.0 PL=0
MOVL C00910 V=800.0 PL=0
MOVL C00911 V=800.0 PL=0
MOVL C00912 V=800.0 PL=0
MOVL C00913 V=800.0 PL=0
MOVL C00914 V=800.0 PL=0
MOVL C00915 V=800.0 PL=0
MOVL C00916 V=800.0 PL=0
MOVL C00917 V=800.0 PL=0
MOVL C00918 V=800.0 PL=0
MOVL C00919 V=800.0 PL=0
MOVL C00920 V=800.0 PL=0
MOVL C00921 V=800.0 PL=0
MOVL C00922 V=800.0 PL=0
MOVL C00923 V=800.0 PL=0
MOVL C00924 V=800.0 PL=0
MOVL C00925 V=800.0 PL=0
MOVL C00926 V=800.0 PL=0
MOVL C00927 V=800.0 PL=0
MOVL C00928 V=800.0 PL=0
MOVL C00929 V=800.0 PL=0
MOVL C00930 V=800.0 PL=0
MOVL C00931 V=800.0 PL=0
MOVL C00932 V=800.0 PL=0
MOVL C00933 V=800.0 PL=0
MOVL C00934 V=800.0 PL=0
MOVL C00935 V=800.0 PL=0
MOVL C00936 V=800.0 PL=0
MOVL C00937 V=800.0 PL=0
MOVL C00938 V=800.0 PL=0
MOVL C00939 V=800.0 PL=0
MOVL C00940 V=800.0 PL=0
MOVL C00941 V=800.0 PL=0
MOVL C00942 V=800.0 PL=0
MOVL C00943 V=800.0 PL=0
MOVL C00944 V=800.0 PL=0
MOVL C00945 V=800.0 PL=0
MOVL C00946 V=800.0 PL=0
MOVL C00947 V=800.0 PL=0
MOVL C00948 V=800.0 PL=0
MOVL C00949 V=800.0 PL=0
MOVL C00950 V=800.0 PL=0
MOVL C00951 V=800.0 PL=0
MOVL C00952 V=800.0 PL=0
MOVL C00953 V=800.0 PL=0
MOVL C00954 V=800.0 PL=0
MOVL C00955 V=800.0 PL=0
MOVL C00956 V=800.0 PL=0
MOVL C00957 V=800.0 PL=0
MOVL C00958 V=800.0 PL=0
MOVL C00959 V=800.0 PL=0
MOVL C00960 V=800.0 PL=0
MOVL C00961 V=800.0 PL=0
MOVL C00962 V=800.0 PL=0
MOVL C00963 V=800.0 PL=0
MOVL C00964 V=800.0 PL=0
MOVL C00965 V=800.0 PL=0
MOVL C00966 V=800.0 PL=0
MOVL C00967 V=800.0 PL=0
MOVL C00968 V=800.0 PL=0
MOVL C00969 V=800.0 PL=0
MOVL C00970 V=800.0 PL=0
MOVL C00971 V=800.0 PL=0
MOVL C00972 V=800.0 PL=0
MOVL C00973 V=800.0 PL=0
MOVL C00974 V=800.0 PL=0
MOVL C00975 V=800.0 PL=0
MOVL C00976 V=800.0 PL=0
MOVL C00977 V=800.0 PL=0
MOVL C00978 V=800.0 PL=0
MOVL C00979 V=800.0 PL=0
MOVL C00980 V=800.0 PL=0
MOVL C00981 V=800.0 PL=0
MOVL C00982 V=800.0 PL=0
MOVL C00983 V=800.0 PL=0
MOVL C00984 V=800.0 PL=0
MOVL C00985 V=800.0 PL=0
MOVL C00986 V=800.0 PL=0
MOVL C00987 V=800.0 PL=0
MOVL C00988 V=800.0 PL=0
MOVL C00989 V=800.0 PL=0
MOVL C00990 V=800.0 PL=0
MOVL C00991 V=800.0 PL=0
MOVL C00992 V=800.0 PL=0
MOVL C00993 V=800.0 PL=0
MOVL C00994 V=800.0 PL=0
MOVL C00995 V=800.0 PL=0
MOVL C00996 V=800.0 PL=0
MOVL C00997 V=800.0 PL=0
MOVL C00998 V=800.0 PL=0
MOVL C00999 V=800.0 PL=0
MOVL C01000 V=800.0 PL=0
MOVL C01001 V=800.0 PL=0
MOVL C01002 V=800.0 PL=0
MOVL C01003 V=800.0 PL=0
MOVL C01004 V=800.0 PL=0
MOVL C01005 V=800.0 PL=0
MOVL C01006 V=800.0 PL=0
MOVL C01007 V=800.0 PL=0
MOVL C01008 V=800.0 PL=0
MOVL C01009 V=800.0 PL=0
MOVL C01010 V=800.0 PL=0
MOVL C01011 V=800.0 PL=0
MOVL C01012 V=800.0 PL=0
MOVL C01013 V=800.0 PL=0
MOVL C01014 V=800.0 PL=0
MOVL C01015 V=800.0 PL=0
MOVL C01016 V=800.0 PL=0
MOVL C01017 V=800.0 PL=0
MOVL C01018 V=800.0 PL=0
MOVL C01019 V=800.0 PL=0
MOVL C01020 V=800.0 PL=0
MOVL C01021 V=800.0 PL=0
MOVL C01022 V=800.0 PL=0
MOVL C01023 V=800.0 PL=0
MOVL C01024 V=800.0 PL=0
MOVL C01025 V=800.0 PL=0
MOVL C01026 V=800.0 PL=0
MOVL C01027 V=800.0 PL=0
MOVL C01028 V=800.0 PL=0
MOVL C01029 V=800.0 PL=0
MOVL C01030 V=800.0 PL=0
MOVL C01031 V=800.0 PL=0
MOVL C01032 V=800.0 PL=0
MOVL C01033 V=800.0 PL=0
MOVL C01034 V=800.0 PL=0
MOVL C01035 V=800.0 PL=0
MOVL C01036 V=800.0 PL=0
MOVL C01037 V=800.0 PL=0
MOVL C01038 V=800.0 PL=0
MOVL C01039 V=800.0 PL=0
MOVL C01040 V=800.0 PL=0
MOVL C01041 V=800.0 PL=0
MOVL C01042 V=800.0 PL=0
MOVL C01043 V=800.0 PL=0
MOVL C01044 V=800.0 PL=0
MOVL C01045 V=800.0 PL=0
MOVL C01046 V=800.0 PL=0
MOVL C01047 V=800.0 PL=0
MOVL C01048 V=800.0 PL=0
MOVL C01049 V=800.0 PL=0
MOVL C01050 V=800.0 PL=0
MOVL C01051 V=800.0 PL=0
MOVL C01052 V=800.0 PL=0
MOVL C01053 V=800.0 PL=0
MOVL C01054 V=800.0 PL=0
MOVL C01055 V=800.0 PL=0
MOVL C01056 V=800.0 PL=0
MOVL C01057 V=800.0 PL=0
MOVL C01058 V=800.0 PL=0
MOVL C01059 V=800.0 PL=0
MOVL C01060 V=800.0 PL=0
MOVL C01061 V=800.0 PL=0
MOVL C01062 V=800.0 PL=0
MOVL C01063 V=800.0 PL=0
MOVL C01064 V=800.0 PL=0
MOVL C01065 V=800.0 PL=0
MOVL C01066 V=800.0 PL=0
MOVL C01067 V=800.0 PL=0
MOVL C01068 V=800.0 PL=0
MOVL C01069 V=800.0 PL=0
MOVL C01070 V=800.0 PL=0
MOVL C01071 V=800.0 PL=0
MOVL C01072 V=800.0 PL=0
MOVL C01073 V=800.0 PL=0
MOVL C01074 V=800.0 PL=0
MOVL C01075 V=800.0 PL=0
MOVL C01076 V=800.0 PL=0
MOVL C01077 V=800.0 PL=0
MOVL C01078 V=800.0 PL=0
MOVL C01079 V=800.0 PL=0
MOVL C01080 V=800.0 PL=0
MOVL C01081 V=800.0 PL=0
MOVL C01082 V=800.0 PL=0
MOVL C01083 V=800.0 PL=0
MOVL C01084 V=800.0 PL=0
MOVL C01085 V=800.0 PL=0
MOVL C01086 V=800.0 PL=0
MOVL C01087 V=800.0 PL=0
MOVL C01088 V=800.0 PL=0
MOVL C01089 V=800.0 PL=0
MOVL C01090 V=800.0 PL=0
MOVL C01091 V=800.0 PL=0
MOVL C01092 V=800.0 PL=0
MOVL C01093 V=800.0 PL=0
MOVL C01094 V=800.0 PL=0
MOVL C01095 V=800.0 PL=0
MOVL C01096 V=800.0 PL=0
MOVL C01097 V=800.0 PL=0
MOVL C01098 V=800.0 PL=0
MOVL C01099 V=800.0 PL=0
MOVL C01100 V=800.0 PL=0
MOVL C01101 V=800.0 PL=0
MOVL C01102 V=800.0 PL=0
MOVL C01103 V=800.0 PL=0
MOVL C01104 V=800.0 PL=0
MOVL C01105 V=800.0 PL=0
MOVL C01106 V=800.0 PL=0
MOVL C01107 V=800.0 PL=0
MOVL C01108 V=800.0 PL=0
MOVL C01109 V=800.0 PL=0
MOVL C01110 V=800.0 PL=0
MOVL C01111 V=800.0 PL=0
MOVL C01112 V=800.0 PL=0
MOVL C01113 V=800.0 PL=0
MOVL C01114 V=800.0 PL=0
MOVL C01115 V=800.0 PL=0
MOVL C01116 V=800.0 PL=0
MOVL C01117 V=800.0 PL=0
MOVL C01118 V=800.0 PL=0
MOVL C01119 V=800.0 PL=0
MOVL C01120 V=800.0 PL=0
MOVL C01121 V=800.0 PL=0
MOVL C01122 V=800.0 PL=0
MOVL C01123 V=800.0 PL=0
MOVL C01124 V=800.0 PL=0
MOVL C01125 V=800.0 PL=0
MOVL C01126 V=800.0 PL=0
MOVL C01127 V=800.0 PL=0
MOVL C01128 V=800.0 PL=0
MOVL C01129 V=800.0 PL=0
MOVL C01130 V=800.0 PL=0
MOVL C01131 V=800.0 PL=0
MOVL C01132 V=800.0 PL=0
MOVL C01133 V=800.0 PL=0
MOVL C01134 V=800.0 PL=0
MOVL C01135 V=800.0 PL=0
MOVL C01136 V=800.0 PL=0
MOVL C01137 V=800.0 PL=0
MOVL C01138 V=800.0 PL=0
MOVL C01139 V=800.0 PL=0
MOVL C01140 V=800.0 PL=0
MOVL C01141 V=800.0 PL=0
MOVL C01142 V=800.0 PL=0
MOVL C01143 V=800.0 PL=0
MOVL C01144 V=800.0 PL=0
MOVL C01145 V=800.0 PL=0
MOVL C01146 V=800.0 PL=0
MOVL C01147 V=800.0 PL=0
MOVL C01148 V=800.0 PL=0
MOVL C01149 V=800.0 PL=0
MOVL C01150 V=800.0 PL=0
MOVL C01151 V=800.0 PL=0
MOVL C01152 V=800.0 PL=0
MOVL C01153 V=800.0 PL=0
MOVL C01154 V=800.0 PL=0
MOVL C01155 V=800.0 PL=0
MOVL C01156 V=800.0 PL=0
MOVL C01157 V=800.0 PL=0
MOVL C01158 V=800.0 PL=0
MOVL C01159 V=800.0 PL=0
MOVL C01160 V=800.0 PL=0
MOVL C01161 V=800.0 PL=0
MOVL C01162 V=800.0 PL=0
MOVL C01163 V=800.0 PL=0
MOVL C01164 V=800.0 PL=0
MOVL C01165 V=800.0 PL=0
MOVL C01166 V=800.0 PL=0
MOVL C01167 V=800.0 PL=0
MOVL C01168 V=800.0 PL=0
MOVL C01169 V=800.0 PL=0
MOVL C01170 V=800.0 PL=0
MOVL C01171 V=800.0 PL=0
MOVL C01172 V=800.0 PL=0
MOVL C01173 V=800.0 PL=0
MOVL C01174 V=800.0 PL=0
MOVL C01175 V=800.0 PL=0
MOVL C01176 V=800.0 PL=0
MOVL C01177 V=800.0 PL=0
MOVL C01178 V=800.0 PL=0
MOVL C01179 V=800.0 PL=0
MOVL C01180 V=800.0 PL=0
MOVL C01181 V=800.0 PL=0
MOVL C01182 V=800.0 PL=0
MOVL C01183 V=800.0 PL=0
MOVL C01184 V=800.0 PL=0
MOVL C01185 V=800.0 PL=0
MOVL C01186 V=800.0 PL=0
MOVL C01187 V=800.0 PL=0
MOVL C01188 V=800.0 PL=0
MOVL C01189 V=800.0 PL=0
MOVL C01190 V=800.0 PL=0
MOVL C01191 V=800.0 PL=0
MOVL C01192 V=800.0 PL=0
MOVL C01193 V=800.0 PL=0
MOVL C01194 V=800.0 PL=0
MOVL C01195 V=800.0 PL=0
MOVL C01196 V=800.0 PL=0
MOVL C01197 V=800.0 PL=0
MOVL C01198 V=800.0 PL=0
MOVL C01199 V=800.0 PL=0
MOVL C01200 V=800.0 PL=0
MOVL C01201 V=800.0 PL=0
MOVL C01202 V=800.0 PL=0
MOVL C01203 V=800.0 PL=0
MOVL C01204 V=800.0 PL=0
MOVL C01205 V=800.0 PL=0
MOVL C01206 V=800.0 PL=0
MOVL C01207 V=800.0 PL=0
MOVL C01208 V=800.0 PL=0
MOVL C01209 V=800.0 PL=0
MOVL C01210 V=800.0 PL=0
MOVL C01211 V=800.0 PL=0
MOVL C01212 V=800.0 PL=0
MOVL C01213 V=800.0 PL=0
MOVL C01214 V=800.0 PL=0
MOVL C01215 V=800.0 PL=0
MOVL C01216 V=800.0 PL=0
MOVL C01217 V=800.0 PL=0
MOVL C01218 V=800.0 PL=0
MOVL C01219 V=800.0 PL=0
MOVL C01220 V=800.0 PL=0
MOVL C01221 V=800.0 PL=0
MOVL C01222 V=800.0 PL=0
MOVL C01223 V=800.0 PL=0
MOVL C01224 V=800.0 PL=0
MOVL C01225 V=800.0 PL=0
MOVL C01226 V=800.0 PL=0
MOVL C01227 V=800.0 PL=0
MOVL C01228 V=800.0 PL=0
MOVL C01229 V=800.0 PL=0
MOVL C01230 V=800.0 PL=0
MOVL C01231 V=800.0 PL=0
MOVL C01232 V=800.0 PL=0
MOVL C01233 V=800.0 PL=0
MOVL C01234 V=800.0 PL=0
MOVL C01235 V=800.0 PL=0
MOVL C01236 V=800.0 PL=0
MOVL C01237 V=800.0 PL=0
MOVL C01238 V=800.0 PL=0
MOVL C01239 V=800.0 PL=0
MOVL C01240 V=800.0 PL=0
MOVL C01241 V=800.0 PL=0
MOVL C01242 V=800.0 PL=0
MOVL C01243 V=800.0 PL=0
MOVL C01244 V=800.0 PL=0
MOVL C01245 V=800.0 PL=0
MOVL C01246 V=800.0 PL=0
MOVL C01247 V=800.0 PL=0
MOVL C01248 V=800.0 PL=0
MOVL C01249 V=800.0 PL=0
MOVL C01250 V=800.0 PL=0
MOVL C01251 V=800.0 PL=0
MOVL C01252 V=800.0 PL=0
MOVL C01253 V=800.0 PL=0
MOVL C01254 V=800.0 PL=0
MOVL C01255 V=800.0 PL=0
MOVL C01256 V=800.0 PL=0
MOVL C01257 V=800.0 PL=0
MOVL C01258 V=800.0 PL=0
MOVL C01259 V=800.0 PL=0
MOVL C01260 V=800.0 PL=0
MOVL C01261 V=800.0 PL=0
MOVL C01262 V=800.0 PL=0
MOVL C01263 V=800.0 PL=0
MOVL C01264 V=800.0 PL=0
MOVL C01265 V=800.0 PL=0
MOVL C01266 V=800.0 PL=0
MOVL C01267 V=800.0 PL=0
MOVL C01268 V=800.0 PL=0
MOVL C01269 V=800.0 PL=0
MOVL C01270 V=800.0 PL=0
MOVL C01271 V=800.0 PL=0
MOVL C01272 V=800.0 PL=0
MOVL C01273 V=800.0 PL=0
MOVL C01274 V=800.0 PL=0
MOVL C01275 V=800.0 PL=0
MOVL C01276 V=800.0 PL=0
MOVL C01277 V=800.0 PL=0
MOVL C01278 V=800.0 PL=0
MOVL C01279 V=800.0 PL=0
MOVL C01280 V=800.0 PL=0
MOVL C01281 V=800.0 PL=0
MOVL C01282 V=800.0 PL=0
MOVL C01283 V=800.0 PL=0
MOVL C01284 V=800.0 PL=0
MOVL C01285 V=800.0 PL=0
MOVL C01286 V=800.0 PL=0
MOVL C01287 V=800.0 PL=0
MOVL C01288 V=800.0 PL=0
MOVL C01289 V=800.0 PL=0
MOVL C01290 V=800.0 PL=0
MOVL C01291 V=800.0 PL=0
MOVL C01292 V=800.0 PL=0
MOVL C01293 V=800.0 PL=0
MOVL C01294 V=800.0 PL=0
MOVL C01295 V=800.0 PL=0
MOVL C01296 V=800.0 PL=0
MOVL C01297 V=800.0 PL=0
MOVL C01298 V=800.0 PL=0
MOVL C01299 V=800.0 PL=0
MOVL C01300 V=800.0 PL=0
MOVL C01301 V=800.0 PL=0
MOVL C01302 V=800.0 PL=0
MOVL C01303 V=800.0 PL=0
MOVL C01304 V=800.0 PL=0
MOVL C01305 V=800.0 PL=0
MOVL C01306 V=800.0 PL=0
MOVL C01307 V=800.0 PL=0
MOVL C01308 V=800.0 PL=0
MOVL C01309 V=800.0 PL=0
MOVL C01310 V=800.0 PL=0
MOVL C01311 V=800.0 PL=0
MOVL C01312 V=800.0 PL=0
MOVL C01313 V=800.0 PL=0
MOVL C01314 V=800.0 PL=0
MOVL C01315 V=800.0 PL=0
MOVL C01316 V=800.0 PL=0
MOVL C01317 V=800.0 PL=0
MOVL C01318 V=800.0 PL=0
MOVL C01319 V=800.0 PL=0
MOVL C01320 V=800.0 PL=0
MOVL C01321 V=800.0 PL=0
MOVL C01322 V=800.0 PL=0
MOVL C01323 V=800.0 PL=0
MOVL C01324 V=800.0 PL=0
MOVL C01325 V=800.0 PL=0
MOVL C01326 V=800.0 PL=0
MOVL C01327 V=800.0 PL=0
MOVL C01328 V=800.0 PL=0
MOVL C01329 V=800.0 PL=0
MOVL C01330 V=800.0 PL=0
MOVL C01331 V=800.0 PL=0
MOVL C01332 V=800.0 PL=0
MOVL C01333 V=800.0 PL=0
MOVL C01334 V=800.0 PL=0
MOVL C01335 V=800.0 PL=0
MOVL C01336 V=800.0 PL=0
MOVL C01337 V=800.0 PL=0
MOVL C01338 V=800.0 PL=0
MOVL C01339 V=800.0 PL=0
MOVL C01340 V=800.0 PL=0
MOVL C01341 V=800.0 PL=0
MOVL C01342 V=800.0 PL=0
MOVL C01343 V=800.0 PL=0
MOVL C01344 V=800.0 PL=0
MOVL C01345 V=800.0 PL=0
MOVL C01346 V=800.0 PL=0
MOVL C01347 V=800.0 PL=0
MOVL C01348 V=800.0 PL=0
MOVL C01349 V=800.0 PL=0
MOVL C01350 V=800.0 PL=0
MOVL C01351 V=800.0 PL=0
MOVL C01352 V=800.0 PL=0
MOVL C01353 V=800.0 PL=0
MOVL C01354 V=800.0 PL=0
MOVL C01355 V=800.0 PL=0
MOVL C01356 V=800.0 PL=0
MOVL C01357 V=800.0 PL=0
MOVL C01358 V=800.0 PL=0
MOVL C01359 V=800.0 PL=0
MOVL C01360 V=800.0 PL=0
MOVL C01361 V=800.0 PL=0
MOVL C01362 V=800.0 PL=0
MOVL C01363 V=800.0 PL=0
MOVL C01364 V=800.0 PL=0
MOVL C01365 V=800.0 PL=0
MOVL C01366 V=800.0 PL=0
MOVL C01367 V=800.0 PL=0
MOVL C01368 V=800.0 PL=0
MOVL C01369 V=800.0 PL=0
MOVL C01370 V=800.0 PL=0
MOVL C01371 V=800.0 PL=0
MOVL C01372 V=800.0 PL=0
MOVL C01373 V=800.0 PL=0
MOVL C01374 V=800.0 PL=0
MOVL C01375 V=800.0 PL=0
MOVL C01376 V=800.0 PL=0
MOVL C01377 V=800.0 PL=0
MOVL C01378 V=800.0 PL=0
MOVL C01379 V=800.0 PL=0
MOVL C01380 V=800.0 PL=0
MOVL C01381 V=800.0 PL=0
MOVL C01382 V=800.0 PL=0
MOVL C01383 V=800.0 PL=0
MOVL C01384 V=800.0 PL=0
MOVL C01385 V=800.0 PL=0
MOVL C01386 V=800.0 PL=0
MOVL C01387 V=800.0 PL=0
MOVL C01388 V=800.0 PL=0
MOVL C01389 V=800.0 PL=0
MOVL C01390 V=800.0 PL=0
MOVL C01391 V=800.0 PL=0
MOVL C01392 V=800.0 PL=0
MOVL C01393 V=800.0 PL=0
MOVL C01394 V=800.0 PL=0
MOVL C01395 V=800.0 PL=0
MOVL C01396 V=800.0 PL=0
MOVL C01397 V=800.0 PL=0
MOVL C01398 V=800.0 PL=0
MOVL C01399 V=800.0 PL=0
MOVL C01400 V=800.0 PL=0
MOVL C01401 V=800.0 PL=0
MOVL C01402 V=800.0 PL=0
MOVL C01403 V=800.0 PL=0
MOVL C01404 V=800.0 PL=0
MOVL C01405 V=800.0 PL=0
MOVL C01406 V=800.0 PL=0
MOVL C01407 V=800.0 PL=0
MOVL C01408 V=800.0 PL=0
MOVL C01409 V=800.0 PL=0
MOVL C01410 V=800.0 PL=0
MOVL C01411 V=800.0 PL=0
MOVL C01412 V=800.0 PL=0
MOVL C01413 V=800.0 PL=0
MOVL C01414 V=800.0 PL=0
MOVL C01415 V=800.0 PL=0
MOVL C01416 V=800.0 PL=0
MOVL C01417 V=800.0 PL=0
MOVL C01418 V=800.0 PL=0
MOVL C01419 V=800.0 PL=0
MOVL C01420 V=800.0 PL=0
MOVL C01421 V=800.0 PL=0
MOVL C01422 V=800.0 PL=0
MOVL C01423 V=800.0 PL=0
MOVL C01424 V=800.0 PL=0
MOVL C01425 V=800.0 PL=0
MOVL C01426 V=800.0 PL=0
MOVL C01427 V=800.0 PL=0
MOVL C01428 V=800.0 PL=0
MOVL C01429 V=800.0 PL=0
MOVL C01430 V=800.0 PL=0
MOVL C01431 V=800.0 PL=0
MOVL C01432 V=800.0 PL=0
MOVL C01433 V=800.0 PL=0
MOVL C01434 V=800.0 PL=0
MOVL C01435 V=800.0 PL=0
MOVL C01436 V=800.0 PL=0
MOVL C01437 V=800.0 PL=0
MOVL C01438 V=800.0 PL=0
MOVL C01439 V=800.0 PL=0
MOVL C01440 V=800.0 PL=0
MOVL C01441 V=800.0 PL=0
MOVL C01442 V=800.0 PL=0
MOVL C01443 V=800.0 PL=0
MOVL C01444 V=800.0 PL=0
MOVL C01445 V=800.0 PL=0
MOVL C01446 V=800.0 PL=0
MOVL C01447 V=800.0 PL=0
MOVL C01448 V=800.0 PL=0
MOVL C01449 V=800.0 PL=0
MOVL C01450 V=800.0 PL=0
MOVL C01451 V=800.0 PL=0
MOVL C01452 V=800.0 PL=0
MOVL C01453 V=800.0 PL=0
MOVL C01454 V=800.0 PL=0
MOVL C01455 V=800.0 PL=0
MOVL C01456 V=800.0 PL=0
MOVL C01457 V=800.0 PL=0
MOVL C01458 V=800.0 PL=0
MOVL C01459 V=800.0 PL=0
MOVL C01460 V=800.0 PL=0
MOVL C01461 V=800.0 PL=0
MOVL C01462 V=800.0 PL=0
MOVL C01463 V=800.0 PL=0
MOVL C01464 V=800.0 PL=0
MOVL C01465 V=800.0 PL=0
MOVL C01466 V=800.0 PL=0
MOVL C01467 V=800.0 PL=0
MOVL C01468 V=800.0 PL=0
MOVL C01469 V=800.0 PL=0
MOVL C01470 V=800.0 PL=0
MOVL C01471 V=800.0 PL=0
MOVL C01472 V=800.0 PL=0
MOVL C01473 V=800.0 PL=0
MOVL C01474 V=800.0 PL=0
MOVL C01475 V=800.0 PL=0
MOVL C01476 V=800.0 PL=0
MOVL C01477 V=800.0 PL=0
MOVL C01478 V=800.0 PL=0
MOVL C01479 V=800.0 PL=0
MOVL C01480 V=800.0 PL=0
MOVL C01481 V=800.0 PL=0
MOVL C01482 V=800.0 PL=0
MOVL C01483 V=800.0 PL=0
MOVL C01484 V=800.0 PL=0
MOVL C01485 V=800.0 PL=0
MOVL C01486 V=800.0 PL=0
MOVL C01487 V=800.0 PL=0
MOVL C01488 V=800.0 PL=0
MOVL C01489 V=800.0 PL=0
MOVL C01490 V=800.0 PL=0
MOVL C01491 V=800.0 PL=0
MOVL C01492 V=800.0 PL=0
MOVL C01493 V=800.0 PL=0
MOVL C01494 V=800.0 PL=0
MOVL C01495 V=800.0 PL=0
MOVL C01496 V=800.0 PL=0
MOVL C01497 V=800.0 PL=0
MOVL C01498 V=800.0 PL=0
MOVL C01499 V=800.0 PL=0
MOVL C01500 V=800.0 PL=0
MOVL C01501 V=800.0 PL=0
MOVL C01502 V=800.0 PL=0
MOVL C01503 V=800.0 PL=0
MOVL C01504 V=800.0 PL=0
MOVL C01505 V=800.0 PL=0
MOVL C01506 V=800.0 PL=0
MOVL C01507 V=800.0 PL=0
MOVL C01508 V=800.0 PL=0
MOVL C01509 V=800.0 PL=0
MOVL C01510 V=800.0 PL=0
MOVL C01511 V=800.0 PL=0
MOVL C01512 V=800.0 PL=0
MOVL C01513 V=800.0 PL=0
MOVL C01514 V=800.0 PL=0
MOVL C01515 V=800.0 PL=0
MOVL C01516 V=800.0 PL=0
MOVL C01517 V=800.0 PL=0
MOVL C01518 V=800.0 PL=0
MOVL C01519 V=800.0 PL=0
MOVL C01520 V=800.0 PL=0
MOVL C01521 V=800.0 PL=0
MOVL C01522 V=800.0 PL=0
MOVL C01523 V=800.0 PL=0
MOVL C01524 V=800.0 PL=0
MOVL C01525 V=800.0 PL=0
MOVL C01526 V=800.0 PL=0
MOVL C01527 V=800.0 PL=0
MOVL C01528 V=800.0 PL=0
MOVL C01529 V=800.0 PL=0
MOVL C01530 V=800.0 PL=0
MOVL C01531 V=800.0 PL=0
MOVL C01532 V=800.0 PL=0
MOVL C01533 V=800.0 PL=0
MOVL C01534 V=800.0 PL=0
MOVL C01535 V=800.0 PL=0
MOVL C01536 V=800.0 PL=0
MOVL C01537 V=800.0 PL=0
MOVL C01538 V=800.0 PL=0
MOVL C01539 V=800.0 PL=0
MOVL C01540 V=800.0 PL=0
MOVL C01541 V=800.0 PL=0
MOVL C01542 V=800.0 PL=0
MOVL C01543 V=800.0 PL=0
MOVL C01544 V=800.0 PL=0
MOVL C01545 V=800.0 PL=0
MOVL C01546 V=800.0 PL=0
MOVL C01547 V=800.0 PL=0
MOVL C01548 V=800.0 PL=0
MOVL C01549 V=800.0 PL=0
MOVL C01550 V=800.0 PL=0
MOVL C01551 V=800.0 PL=0
MOVL C01552 V=800.0 PL=0
MOVL C01553 V=800.0 PL=0
MOVL C01554 V=800.0 PL=0
MOVL C01555 V=800.0 PL=0
MOVL C01556 V=800.0 PL=0
MOVL C01557 V=800.0 PL=0
MOVL C01558 V=800.0 PL=0
MOVL C01559 V=800.0 PL=0
MOVL C01560 V=800.0 PL=0
MOVL C01561 V=800.0 PL=0
MOVL C01562 V=800.0 PL=0
MOVL C01563 V=800.0 PL=0
MOVL C01564 V=800.0 PL=0
MOVL C01565 V=800.0 PL=0
MOVL C01566 V=800.0 PL=0
MOVL C01567 V=800.0 PL=0
MOVL C01568 V=800.0 PL=0
MOVL C01569 V=800.0 PL=0
MOVL C01570 V=800.0 PL=0
MOVL C01571 V=800.0 PL=0
MOVL C01572 V=800.0 PL=0
MOVL C01573 V=800.0 PL=0
MOVL C01574 V=800.0 PL=0
MOVL C01575 V=800.0 PL=0
MOVL C01576 V=800.0 PL=0
MOVL C01577 V=800.0 PL=0
MOVL C01578 V=800.0 PL=0
MOVL C01579 V=800.0 PL=0
MOVL C01580 V=800.0 PL=0
MOVL C01581 V=800.0 PL=0
MOVL C01582 V=800.0 PL=0
MOVL C01583 V=800.0 PL=0
MOVL C01584 V=800.0 PL=0
MOVL C01585 V=800.0 PL=0
MOVL C01586 V=800.0 PL=0
MOVL C01587 V=800.0 PL=0
MOVL C01588 V=800.0 PL=0
MOVL C01589 V=800.0 PL=0
MOVL C01590 V=800.0 PL=0
MOVL C01591 V=800.0 PL=0
MOVL C01592 V=800.0 PL=0
MOVL C01593 V=800.0 PL=0
MOVL C01594 V=800.0 PL=0
MOVL C01595 V=800.0 PL=0
MOVL C01596 V=800.0 PL=0
MOVL C01597 V=800.0 PL=0
MOVL C01598 V=800.0 PL=0
MOVL C01599 V=800.0 PL=0
MOVL C01600 V=800.0 PL=0
MOVL C01601 V=800.0 PL=0
MOVL C01602 V=800.0 PL=0
MOVL C01603 V=800.0 PL=0
MOVL C01604 V=800.0 PL=0
MOVL C01605 V=800.0 PL=0
MOVL C01606 V=800.0 PL=0
MOVL C01607 V=800.0 PL=0
MOVL C01608 V=800.0 PL=0
MOVL C01609 V=800.0 PL=0
MOVL C01610 V=800.0 PL=0
MOVL C01611 V=800.0 PL=0
MOVL C01612 V=800.0 PL=0
MOVL C01613 V=800.0 PL=0
MOVL C01614 V=800.0 PL=0
MOVL C01615 V=800.0 PL=0
MOVL C01616 V=800.0 PL=0
MOVL C01617 V=800.0 PL=0
MOVL C01618 V=800.0 PL=0
MOVL C01619 V=800.0 PL=0
MOVL C01620 V=800.0 PL=0
MOVL C01621 V=800.0 PL=0
MOVL C01622 V=800.0 PL=0
MOVL C01623 V=800.0 PL=0
MOVL C01624 V=800.0 PL=0
MOVL C01625 V=800.0 PL=0
MOVL C01626 V=800.0 PL=0
MOVL C01627 V=800.0 PL=0
MOVL C01628 V=800.0 PL=0
MOVL C01629 V=800.0 PL=0
MOVL C01630 V=800.0 PL=0
MOVL C01631 V=800.0 PL=0
MOVL C01632 V=800.0 PL=0
MOVL C01633 V=800.0 PL=0
MOVL C01634 V=800.0 PL=0
MOVL C01635 V=800.0 PL=0
MOVL C01636 V=800.0 PL=0
MOVL C01637 V=800.0 PL=0
MOVL C01638 V=800.0 PL=0
MOVL C01639 V=800.0 PL=0
MOVL C01640 V=800.0 PL=0
MOVL C01641 V=800.0 PL=0
MOVL C01642 V=800.0 PL=0
MOVL C01643 V=800.0 PL=0
MOVL C01644 V=800.0 PL=0
MOVL C01645 V=800.0 PL=0
MOVL C01646 V=800.0 PL=0
MOVL C01647 V=800.0 PL=0
MOVL C01648 V=800.0 PL=0
MOVL C01649 V=800.0 PL=0
MOVL C01650 V=800.0 PL=0
MOVL C01651 V=800.0 PL=0
MOVL C01652 V=800.0 PL=0
MOVL C01653 V=800.0 PL=0
MOVL C01654 V=800.0 PL=0
MOVL C01655 V=800.0 PL=0
MOVL C01656 V=800.0 PL=0
MOVL C01657 V=800.0 PL=0
MOVL C01658 V=800.0 PL=0
MOVL C01659 V=800.0 PL=0
MOVL C01660 V=800.0 PL=0
MOVL C01661 V=800.0 PL=0
MOVL C01662 V=800.0 PL=0
MOVL C01663 V=800.0 PL=0
MOVL C01664 V=800.0 PL=0
MOVL C01665 V=800.0 PL=0
MOVL C01666 V=800.0 PL=0
MOVL C01667 V=800.0 PL=0
MOVL C01668 V=800.0 PL=0
MOVL C01669 V=800.0 PL=0
MOVL C01670 V=800.0 PL=0
MOVL C01671 V=800.0 PL=0
MOVL C01672 V=800.0 PL=0
MOVL C01673 V=800.0 PL=0
MOVL C01674 V=800.0 PL=0
MOVL C01675 V=800.0 PL=0
MOVL C01676 V=800.0 PL=0
MOVL C01677 V=800.0 PL=0
MOVL C01678 V=800.0 PL=0
MOVL C01679 V=800.0 PL=0
MOVL C01680 V=800.0 PL=0
MOVL C01681 V=800.0 PL=0
MOVL C01682 V=800.0 PL=0
MOVL C01683 V=800.0 PL=0
MOVL C01684 V=800.0 PL=0
MOVL C01685 V=800.0 PL=0
MOVL C01686 V=800.0 PL=0
MOVL C01687 V=800.0 PL=0
MOVL C01688 V=800.0 PL=0
MOVL C01689 V=800.0 PL=0
MOVL C01690 V=800.0 PL=0
MOVL C01691 V=800.0 PL=0
MOVL C01692 V=800.0 PL=0
MOVL C01693 V=800.0 PL=0
MOVL C01694 V=800.0 PL=0
MOVL C01695 V=800.0 PL=0
MOVL C01696 V=800.0 PL=0
MOVL C01697 V=800.0 PL=0
MOVL C01698 V=800.0 PL=0
MOVL C01699 V=800.0 PL=0
MOVL C01700 V=800.0 PL=0
MOVL C01701 V=800.0 PL=0
MOVL C01702 V=800.0 PL=0
MOVL C01703 V=800.0 PL=0
MOVL C01704 V=800.0 PL=0
MOVL C01705 V=800.0 PL=0
MOVL C01706 V=800.0 PL=0
MOVL C01707 V=800.0 PL=0
MOVL C01708 V=800.0 PL=0
MOVL C01709 V=800.0 PL=0
MOVL C01710 V=800.0 PL=0
MOVL C01711 V=800.0 PL=0
MOVL C01712 V=800.0 PL=0
MOVL C01713 V=800.0 PL=0
MOVL C01714 V=800.0 PL=0
MOVL C01715 V=800.0 PL=0
MOVL C01716 V=800.0 PL=0
MOVL C01717 V=800.0 PL=0
MOVL C01718 V=800.0 PL=0
MOVL C01719 V=800.0 PL=0
MOVL C01720 V=800.0 PL=0
MOVL C01721 V=800.0 PL=0
MOVL C01722 V=800.0 PL=0
MOVL C01723 V=800.0 PL=0
MOVL C01724 V=800.0 PL=0
MOVL C01725 V=800.0 PL=0
MOVL C01726 V=800.0 PL=0
MOVL C01727 V=800.0 PL=0
MOVL C01728 V=800.0 PL=0
MOVL C01729 V=800.0 PL=0
MOVL C01730 V=800.0 PL=0
MOVL C01731 V=800.0 PL=0
MOVL C01732 V=800.0 PL=0
MOVL C01733 V=800.0 PL=0
MOVL C01734 V=800.0 PL=0
MOVL C01735 V=800.0 PL=0
MOVL C01736 V=800.0 PL=0
MOVL C01737 V=800.0 PL=0
MOVL C01738 V=800.0 PL=0
MOVL C01739 V=800.0 PL=0
MOVL C01740 V=800.0 PL=0
MOVL C01741 V=800.0 PL=0
MOVL C01742 V=800.0 PL=0
MOVL C01743 V=800.0 PL=0
MOVL C01744 V=800.0 PL=0
MOVL C01745 V=800.0 PL=0
MOVL C01746 V=800.0 PL=0
MOVL C01747 V=800.0 PL=0
MOVL C01748 V=800.0 PL=0
MOVL C01749 V=800.0 PL=0
MOVL C01750 V=800.0 PL=0
MOVL C01751 V=800.0 PL=0
MOVL C01752 V=800.0 PL=0
MOVL C01753 V=800.0 PL=0
MOVL C01754 V=800.0 PL=0
MOVL C01755 V=800.0 PL=0
MOVL C01756 V=800.0 PL=0
MOVL C01757 V=800.0 PL=0
MOVL C01758 V=800.0 PL=0
MOVL C01759 V=800.0 PL=0
MOVL C01760 V=800.0 PL=0
MOVL C01761 V=800.0 PL=0
MOVL C01762 V=800.0 PL=0
MOVL C01763 V=800.0 PL=0
MOVL C01764 V=800.0 PL=0
MOVL C01765 V=800.0 PL=0
MOVL C01766 V=800.0 PL=0
MOVL C01767 V=800.0 PL=0
MOVL C01768 V=800.0 PL=0
MOVL C01769 V=800.0 PL=0
MOVL C01770 V=800.0 PL=0
MOVL C01771 V=800.0 PL=0
MOVL C01772 V=800.0 PL=0
MOVL C01773 V=800.0 PL=0
MOVL C01774 V=800.0 PL=0
MOVL C01775 V=800.0 PL=0
MOVL C01776 V=800.0 PL=0
MOVL C01777 V=800.0 PL=0
MOVL C01778 V=800.0 PL=0
MOVL C01779 V=800.0 PL=0
MOVL C01780 V=800.0 PL=0
MOVL C01781 V=800.0 PL=0
MOVL C01782 V=800.0 PL=0
MOVL C01783 V=800.0 PL=0
MOVL C01784 V=800.0 PL=0
MOVL C01785 V=800.0 PL=0
MOVL C01786 V=800.0 PL=0
MOVL C01787 V=800.0 PL=0
MOVL C01788 V=800.0 PL=0
MOVL C01789 V=800.0 PL=0
MOVL C01790 V=800.0 PL=0
MOVL C01791 V=800.0 PL=0
MOVL C01792 V=800.0 PL=0
MOVL C01793 V=800.0 PL=0
MOVL C01794 V=800.0 PL=0
MOVL C01795 V=800.0 PL=0
MOVL C01796 V=800.0 PL=0
MOVL C01797 V=800.0 PL=0
MOVL C01798 V=800.0 PL=0
MOVL C01799 V=800.0 PL=0
MOVL C01800 V=800.0 PL=0
MOVL C01801 V=800.0 PL=0
MOVL C01802 V=800.0 PL=0
MOVL C01803 V=800.0 PL=0
MOVL C01804 V=800.0 PL=0
MOVL C01805 V=800.0 PL=0
MOVL C01806 V=800.0 PL=0
MOVL C01807 V=800.0 PL=0
MOVL C01808 V=800.0 PL=0
MOVL C01809 V=800.0 PL=0
MOVL C01810 V=800.0 PL=0
MOVL C01811 V=800.0 PL=0
MOVL C01812 V=800.0 PL=0
MOVL C01813 V=800.0 PL=0
MOVL C01814 V=800.0 PL=0
MOVL C01815 V=800.0 PL=0
MOVL C01816 V=800.0 PL=0
MOVL C01817 V=800.0 PL=0
MOVL C01818 V=800.0 PL=0
MOVL C01819 V=800.0 PL=0
MOVL C01820 V=800.0 PL=0
MOVL C01821 V=800.0 PL=0
MOVL C01822 V=800.0 PL=0
MOVL C01823 V=800.0 PL=0
MOVL C01824 V=800.0 PL=0
MOVL C01825 V=800.0 PL=0
MOVL C01826 V=800.0 PL=0
MOVL C01827 V=800.0 PL=0
MOVL C01828 V=800.0 PL=0
MOVL C01829 V=800.0 PL=0
MOVL C01830 V=800.0 PL=0
MOVL C01831 V=800.0 PL=0
MOVL C01832 V=800.0 PL=0
MOVL C01833 V=800.0 PL=0
MOVL C01834 V=800.0 PL=0
MOVL C01835 V=800.0 PL=0
MOVL C01836 V=800.0 PL=0
MOVL C01837 V=800.0 PL=0
MOVL C01838 V=800.0 PL=0
MOVL C01839 V=800.0 PL=0
MOVL C01840 V=800.0 PL=0
MOVL C01841 V=800.0 PL=0
MOVL C01842 V=800.0 PL=0
MOVL C01843 V=800.0 PL=0
MOVL C01844 V=800.0 PL=0
MOVL C01845 V=800.0 PL=0
MOVL C01846 V=800.0 PL=0
MOVL C01847 V=800.0 PL=0
MOVL C01848 V=800.0 PL=0
MOVL C01849 V=800.0 PL=0
MOVL C01850 V=800.0 PL=0
MOVL C01851 V=800.0 PL=0
MOVL C01852 V=800.0 PL=0
MOVL C01853 V=800.0 PL=0
MOVL C01854 V=800.0 PL=0
MOVL C01855 V=800.0 PL=0
MOVL C01856 V=800.0 PL=0
MOVL C01857 V=800.0 PL=0
MOVL C01858 V=800.0 PL=0
MOVL C01859 V=800.0 PL=0
MOVL C01860 V=800.0 PL=0
MOVL C01861 V=800.0 PL=0
MOVL C01862 V=800.0 PL=0
MOVL C01863 V=800.0 PL=0
MOVL C01864 V=800.0 PL=0
MOVL C01865 V=800.0 PL=0
MOVL C01866 V=800.0 PL=0
MOVL C01867 V=800.0 PL=0
MOVL C01868 V=800.0 PL=0
MOVL C01869 V=800.0 PL=0
MOVL C01870 V=800.0 PL=0
MOVL C01871 V=800.0 PL=0
MOVL C01872 V=800.0 PL=0
MOVL C01873 V=800.0 PL=0
MOVL C01874 V=800.0 PL=0
MOVL C01875 V=800.0 PL=0
MOVL C01876 V=800.0 PL=0
MOVL C01877 V=800.0 PL=0
MOVL C01878 V=800.0 PL=0
MOVL C01879 V=800.0 PL=0
MOVL C01880 V=800.0 PL=0
MOVL C01881 V=800.0 PL=0
MOVL C01882 V=800.0 PL=0
MOVL C01883 V=800.0 PL=0
MOVL C01884 V=800.0 PL=0
MOVL C01885 V=800.0 PL=0
MOVL C01886 V=800.0 PL=0
MOVL C01887 V=800.0 PL=0
MOVL C01888 V=800.0 PL=0
MOVL C01889 V=800.0 PL=0
MOVL C01890 V=800.0 PL=0
MOVL C01891 V=800.0 PL=0
MOVL C01892 V=800.0 PL=0
MOVL C01893 V=800.0 PL=0
MOVL C01894 V=800.0 PL=0
MOVL C01895 V=800.0 PL=0
MOVL C01896 V=800.0 PL=0
MOVL C01897 V=800.0 PL=0
MOVL C01898 V=800.0 PL=0
MOVL C01899 V=800.0 PL=0
MOVL C01900 V=800.0 PL=0
MOVL C01901 V=800.0 PL=0
MOVL C01902 V=800.0 PL=0
MOVL C01903 V=800.0 PL=0
MOVL C01904 V=800.0 PL=0
MOVL C01905 V=800.0 PL=0
MOVL C01906 V=800.0 PL=0
MOVL C01907 V=800.0 PL=0
MOVL C01908 V=800.0 PL=0
MOVL C01909 V=800.0 PL=0
MOVL C01910 V=800.0 PL=0
MOVL C01911 V=800.0 PL=0
MOVL C01912 V=800.0 PL=0
MOVL C01913 V=800.0 PL=0
MOVL C01914 V=800.0 PL=0
MOVL C01915 V=800.0 PL=0
MOVL C01916 V=800.0 PL=0
MOVL C01917 V=800.0 PL=0
MOVL C01918 V=800.0 PL=0
MOVL C01919 V=800.0 PL=0
MOVL C01920 V=800.0 PL=0
MOVL C01921 V=800.0 PL=0
MOVL C01922 V=800.0 PL=0
MOVL C01923 V=800.0 PL=0
MOVL C01924 V=800.0 PL=0
MOVL C01925 V=800.0 PL=0
MOVL C01926 V=800.0 PL=0
MOVL C01927 V=800.0 PL=0
MOVL C01928 V=800.0 PL=0
MOVL C01929 V=800.0 PL=0
MOVL C01930 V=800.0 PL=0
MOVL C01931 V=800.0 PL=0
MOVL C01932 V=800.0 PL=0
MOVL C01933 V=800.0 PL=0
MOVL C01934 V=800.0 PL=0
MOVL C01935 V=800.0 PL=0
MOVL C01936 V=800.0 PL=0
MOVL C01937 V=800.0 PL=0
MOVL C01938 V=800.0 PL=0
MOVL C01939 V=800.0 PL=0
MOVL C01940 V=800.0 PL=0
MOVL C01941 V=800.0 PL=0
MOVL C01942 V=800.0 PL=0
MOVL C01943 V=800.0 PL=0
MOVL C01944 V=800.0 PL=0
MOVL C01945 V=800.0 PL=0
MOVL C01946 V=800.0 PL=0
MOVL C01947 V=800.0 PL=0
MOVL C01948 V=800.0 PL=0
MOVL C01949 V=800.0 PL=0
MOVL C01950 V=800.0 PL=0
MOVL C01951 V=800.0 PL=0
MOVL C01952 V=800.0 PL=0
MOVL C01953 V=800.0 PL=0
MOVL C01954 V=800.0 PL=0
MOVL C01955 V=800.0 PL=0
MOVL C01956 V=800.0 PL=0
MOVL C01957 V=800.0 PL=0
MOVL C01958 V=800.0 PL=0
MOVL C01959 V=800.0 PL=0
MOVL C01960 V=800.0 PL=0
MOVL C01961 V=800.0 PL=0
MOVL C01962 V=800.0 PL=0
MOVL C01963 V=800.0 PL=0
MOVL C01964 V=800.0 PL=0
MOVL C01965 V=800.0 PL=0
MOVL C01966 V=800.0 PL=0
MOVL C01967 V=800.0 PL=0
MOVL C01968 V=800.0 PL=0
MOVL C01969 V=800.0 PL=0
MOVL C01970 V=800.0 PL=0
MOVL C01971 V=800.0 PL=0
MOVL C01972 V=800.0 PL=0
MOVL C01973 V=800.0 PL=0
MOVL C01974 V=800.0 PL=0
MOVL C01975 V=800.0 PL=0
MOVL C01976 V=800.0 PL=0
MOVL C01977 V=800.0 PL=0
MOVL C01978 V=800.0 PL=0
MOVL C01979 V=800.0 PL=0
MOVL C01980 V=800.0 PL=0
MOVL C01981 V=800.0 PL=0
MOVL C01982 V=800.0 PL=0
MOVL C01983 V=800.0 PL=0
MOVL C01984 V=800.0 PL=0
MOVL C01985 V=800.0 PL=0
MOVL C01986 V=800.0 PL=0
MOVL C01987 V=800.0 PL=0
MOVL C01988 V=800.0 PL=0
MOVL C01989 V=800.0 PL=0
MOVL C01990 V=800.0 PL=0
MOVL C01991 V=800.0 PL=0
MOVL C01992 V=800.0 PL=0
MOVL C01993 V=800.0 PL=0
MOVL C01994 V=800.0 PL=0
MOVL C01995 V=800.0 PL=0
MOVL C01996 V=800.0 PL=0
MOVL C01997 V=800.0 PL=0
MOVL C01998 V=800.0 PL=0
MOVL C01999 V=800.0 PL=0
MOVL C02000 V=800.0 PL=0
MOVL C02001 V=800.0 PL=0
MOVL C02002 V=800.0 PL=0
MOVL C02003 V=800.0 PL=0
MOVL C02004 V=800.0 PL=0
MOVL C02005 V=800.0 PL=0
MOVL C02006 V=800.0 PL=0
MOVL C02007 V=800.0 PL=0
MOVL C02008 V=800.0 PL=0
MOVL C02009 V=800.0 PL=0
MOVL C02010 V=800.0 PL=0
MOVL C02011 V=800.0 PL=0
MOVL C02012 V=800.0 PL=0
MOVL C02013 V=800.0 PL=0
MOVL C02014 V=800.0 PL=0
MOVL C02015 V=800.0 PL=0
MOVL C02016 V=800.0 PL=0
MOVL C02017 V=800.0 PL=0
MOVL C02018 V=800.0 PL=0
MOVL C02019 V=800.0 PL=0
MOVL C02020 V=800.0 PL=0
MOVL C02021 V=800.0 PL=0
MOVL C02022 V=800.0 PL=0
MOVL C02023 V=800.0 PL=0
MOVL C02024 V=800.0 PL=0
MOVL C02025 V=800.0 PL=0
MOVL C02026 V=800.0 PL=0
MOVL C02027 V=800.0 PL=0
MOVL C02028 V=800.0 PL=0
MOVL C02029 V=800.0 PL=0
MOVL C02030 V=800.0 PL=0
MOVL C02031 V=800.0 PL=0
MOVL C02032 V=800.0 PL=0
MOVL C02033 V=800.0 PL=0
MOVL C02034 V=800.0 PL=0
MOVL C02035 V=800.0 PL=0
MOVL C02036 V=800.0 PL=0
MOVL C02037 V=800.0 PL=0
